# B&R Automation Studio project ControlPLC_DataDistribution (part 4)

#### Types.typ
```iecst
TYPE
	Configuration_typ : 	STRUCT
		Exists : BOOL;
		ComPortNumberZaber1Hmi : UINT;
		PyroMultiplicationFactorHmi : REAL;
	END_STRUCT;
	DI_typ : 	STRUCT
		_ : BOOL;
	END_STRUCT;
	DO_typ : 	STRUCT
		_ : BOOL;
	END_STRUCT;
	IO_typ : 	STRUCT
		do : DO_typ;
		di : DI_typ;
	END_STRUCT;
	localInterfaceCommand_typ : 	STRUCT
		exampleCommand : BOOL;
		initializeCalibration : BOOL;
		initializePixel : BOOL;
		capturePixel : BOOL;
		processPixel : BOOL;
		processCalibration : BOOL;
		uploadLUTs : BOOL;
		abort : BOOL;
		uploadTestData : BOOL;
		downloadAndParseTestResults : BOOL;
		initializeOmsTestZaber2 : BOOL;
		initializeOmsTestZaber1 : BOOL;
		setZaber1Pos : BOOL;
		setZaber2PosAndExposure : BOOL;
		checkZaber2Homed : BOOL;
		checkZaber1Homed : BOOL;
		passRequiredMetaData : BOOL;
		passCompleteHandshake : BOOL;
		passAbortedHandshake : BOOL;
		captureFrame : BOOL;
		passAbortedHandshakeWithoutAck : BOOL;
		initializePixelForFrame : BOOL;
	END_STRUCT;
	localInterfaceInternal_typ : 	STRUCT
		PLCOpen : AtnPlcOpenStatus;
		previousState : STATE;
		frameCaptured : BOOL;
		newCommand : BOOL;
		localLockout : BOOL;
		subSystemStatus : ARRAY[0..10]OF STRING[80];
		parameters : localInterfaceParameters_typ;
		missedHeartbeats : USINT;
		lastHeartbeatReceived : INT;
		calibAppNotConnected : BOOL;
		heartbeatTimer : TON;
		cmdTimeoutTimer : TON;
		cmdFrameCaptureTimer : TON;
		homeZaberWaitTimer : TON;
		moveZaberWaitTimer : TON;
		cmdZaberOnWaitTimer : TON;
		pollingAppWaitTimer : TON;
		resultsPollingTimer : TON;
		resultsTimeoutTimer : TON;
		atnPLCOpenCommandParameters : AtnPLCOpenWithParameters;
		atnPLCOpenCommand : AtnPLCOpen;
		measuredPowerList1 : ARRAY[0..100]OF REAL;
		measuredPowerList2 : ARRAY[0..100]OF REAL;
		measuredPowerList3 : ARRAY[0..100]OF REAL;
		measuredPowerList4 : ARRAY[0..100]OF REAL;
		measuredPowerList5 : ARRAY[0..100]OF REAL;
		measuredPowerList6 : ARRAY[0..100]OF REAL;
		measuredPowerList7 : ARRAY[0..100]OF REAL;
		measuredPowerList8 : ARRAY[0..100]OF REAL;
		CommandedPowerList1 : ARRAY[0..100]OF REAL;
		CommandedPowerList2 : ARRAY[0..100]OF REAL;
		CommandedPowerList3 : ARRAY[0..100]OF REAL;
		CommandedPowerList4 : ARRAY[0..100]OF REAL;
		CommandedPowerList5 : ARRAY[0..100]OF REAL;
		CommandedPowerList6 : ARRAY[0..100]OF REAL;
		CommandedPowerList7 : ARRAY[0..100]OF REAL;
		CommandedPowerList8 : ARRAY[0..100]OF REAL;
		LaserTestStatusList1 : ARRAY[0..100]OF STRING[10];
		LaserTestStatusList2 : ARRAY[0..100]OF STRING[10];
		LaserTestStatusList3 : ARRAY[0..100]OF STRING[10];
		LaserTestStatusList4 : ARRAY[0..100]OF STRING[10];
		LaserTestStatusList5 : ARRAY[0..100]OF STRING[10];
		LaserTestStatusList6 : ARRAY[0..100]OF STRING[10];
		LaserTestStatusList7 : ARRAY[0..100]OF STRING[10];
		LaserTestStatusList8 : ARRAY[0..100]OF STRING[10];
		currentPowerLevel : USINT;
		ii : USINT; (*loop variable*)
		appVersionTempString : STRING[5]; (*loop variable*)
	END_STRUCT;
	localInterfaceParameters_typ : 	STRUCT
		uploadLUTs : VFLCRUploadLUTsCmdPars_typ;
		initializePixel : VFLCRInitializePixelCmdPars_typ;
		capturePixel : VFLCRDataCollectionCmdPars_typ;
		adjustZaber1 : VFLCRAdjustZaberAndExpoPars_typ;
		adjustZaber2AndExposure : VFLCRAdjustZaberAndExpoPars_typ;
		initializePixelForFrame : VFLCRInitializePixelCmdPars_typ;
	END_STRUCT;
	localInterfaceStatus_typ : 	STRUCT
		ready : BOOL;
		state : STATE;
		sequence : SEQUENCE;
		calibAppConnected : BOOL;
		processingTestData : BOOL;
		resultsDownloaded : BOOL;
		statusMessage : STRING[vfALARMS_MAX_SNIPPET_STR_LENGTH];
		strStatus : STRING[80];
		LutIdHmi : UDINT;
		AppVersion : STRING[10];
	END_STRUCT;
	localInterface_typ : 	STRUCT
		command : localInterfaceCommand_typ;
		status : localInterfaceStatus_typ;
		internal : localInterfaceInternal_typ;
		parameters : localInterfaceParameters_typ;
	END_STRUCT;
	SEQUENCE :
		(
		SEQUENCE_IDLE,
		SEQUENCE_DONE,
		SEQUENCE_ERROR,
		SEQUENCE_LUT_DELETE,
		SEQUENCE_LUT_FTP,
		SEQUENCE_LUT_TRANSFER,
		SEQUENCE_RESULTS_DOWNLOAD,
		SEQUENCE_RESULTS_PARSE,
		SEQUENCE_MOVE_ZABER2,
		SEQUENCE_MOVE_ZABER1,
		SEQUENCE_OMS_INIT,
		SEQUENCE_OMS_ABORTED,
		SEQUENCE_WAIT_FRAME_CAPTURE
		);
	TEST_MODE :
		(
		TEST_MODE_CONTINUOUS,
		TEST_MODE_SEMI_AUTO
		);
	TEST_RESULT :
		(
		TEST_RESULT_IN_PROGRESS,
		TEST_RESULT_PASSED,
		TEST_RESULT_HIGH_POWER_FAILURE,
		TEST_RESULT_LOW_POWER_FAILURE,
		TEST_RESULT_NO_POWER_FAILURE,
		TEST_RESULT_UNTESTED,
		TEST_RESULT_ABORTED := 10
		);
	STATE :
		(
		STATE_NOT_READY,
		STATE_READY,
		STATE_DONE,
		STATE_ERROR,
		STATE_EXAMPLE_COMMAND,
		STATE_INITIALIZE_CALIBRATION,
		STATE_INITIALIZE_PIXEL,
		STATE_CAPTURE_PIXEL,
		STATE_PROCESS_PIXEL,
		STATE_PROCESS_CALIBRATION,
		STATE_UPLOAD_LUTS,
		STATE_UPLOAD_TEST_DATA,
		STATE_DOWNLOAD_PARSE_RESULTS,
		STATE_INITIALIZE_OMS_TEST_ZABER2,
		STATE_INITIALIZE_OMS_TEST_ZABER1,
		STATE_CHECK_ZABER2_HOMED,
		STATE_CHECK_ZABER1_HOMED,
		STATE_PASS_META_DATA,
		STATE_CAPTURE_FRAME,
		STATE_MOVE_ZABER2_CAM_EXPO,
		STATE_MOVE_ZABER1_CAM,
		STATE_PASS_TEST_COMPLETE,
		STATE_PASS_TEST_ABORTED,
		STATE_PASS_TEST_ABORTED_NO_ACK,
		STATE_INIT_PIXEL_FRAMECAPTURE
		);
END_TYPE
```

#### Variables.var
```iecst
VAR
	IO : IO_typ;
END_VAR
VAR RETAIN
	Configuration : Configuration_typ;
END_VAR
VAR
	task : localInterface_typ;
	logSeqChange_0 : logStateChange;
	logStateChange_0 : logStateChange;
	Name : STRING[80];
	dIn : REFERENCE TO OPCUAData_FROM_Gen3CalibApp_typ;
	dOut : REFERENCE TO OPCUAData_TO_Gen3CalibApp_typ;
	strMachineNumber : STRING[40];
	strFactoryNumber : STRING[40];
END_VAR
VAR CONSTANT
	MAX_MISSED_HEARTBEATS : USINT := 7;
END_VAR
VAR
	activePixelPlaceholder : USINT := 1;
	usingGen3LaserCalibrationApp : BOOL; (*temporary disable*)
END_VAR
```

#### Simulation.st
```iecst
ACTION SimulateIO:

END_ACTION
```

### Program Logical/ProcessControl/VFLCR/VFPTR_System (IEC)

#### Main.st - Init, cyclic, exit code
```iecst
PROGRAM _INIT

	IO.do.counterReset := TRUE;

	subscribePLCOpen(gVFLCR.command.enableModulation,  'VFPTR_System', task.command.enableModulation,  task.internal.PLCOpenEnableModulation);
	subscribePLCOpen(gVFLCR.command.disableModulation, 'VFPTR_System', task.command.disableModulation, task.internal.PLCOpenDisableModulation);

	subscribePLCOpen(gVFLCR.command.openLayer, 'VFPTR_System', task.command.pulseCounterReset, task.internal.PLCOpenCounterReset);
	subscribePLCOpen(gVFLCR.command.abortLayer, 'VFPTR_System', task.command.endTrajectory, task.internal.PLCOpenTrajectory);

	registerStateBool(gVFLCR.inhibit.autoModulation, 'VFPTR_System', task.status.counterResetEnabled);

	registerStateBool(gVFLCR.status.counterResetEnabled, 'VFPTR_System', task.status.counterResetEnabled);
	registerStateBool(gVFLCR.status.modulationEnabled, 'VFPTR_System', task.status.modulationEnabled);
	registerStateBool(gVFLCR.status.userModulationEnabled, 'VFPTR_System', task.status.userModulationEnabled);
	registerStateBool(gVFLCR.status.encoderXSelected, 'VFPTR_System', task.status.encoderXSelected);
	registerStateBool(gVFLCR.status.prepareTrajectory, 'VFPTR_System', task.status.prepareTrajectory);

	// Set timeout
	task.internal.openLayerTON.PT := T#5s;

	// Initialize the lag error statistics function block moving window length.
	FOR i := 0 TO MONITOR_AXIS_MAI BY 1 DO
		task.internal.lagErrorStatistics[i].Enable := TRUE;
		task.internal.lagErrorStatistics[i].Update := TRUE;
		task.internal.lagErrorStatistics[i].MovingWindowLength := Configuration.lagMovingAvgWindowLength;
		task.internal.lagErrorStatistics[i].In := 0.0;
		task.internal.lagErrorStatistics[i]();
	END_FOR

END_PROGRAM

PROGRAM _CYCLIC

	//PiperModuleInterface;

	// Modulation in manual mode requires:
	// - safety interlock reset
	// 		- inhibit probably set elsewhere
	// - modulationEnable flag (set by user)
	// Modulation in auto mode additionally requires:
	// - prepareTrajectory (M-flag)
	// - NOT counterReset (command, maybe also M-flag related?)
	// - build info valid
	// 		- inhibit set elsewhere
	// - CNC gantry group is in GroupStateMoving
	// 		- inhibit set elsewhere
	// - master axis homed and within build volume bounds (+/- 25mm?)
	// 		- inhibit set elsewhere

	// do.enableModulation should be TRUE only while over the build plate; other conditions apply, see above
	// do.counterReset should be FALSE while in a trajectory, TRUE otherwise. Additionally, a positive edge is required after opening a layer and before starting the first trajectory.
	// do.selectEncoderX should be TRUE while printing in the X direction and FALSE while printing in the Y direction (while not lasing, its value is benign)

	///////////////////////////////////////////////////////////////
	// API:
	//	Requires:
	//	- nothing
	//	Commands:
	//	- enableModulation 			- Allows the lasers to fire
	//	- disableModulation 		- Prevents the lasers from firing
	//  Statuses:
	//	- modulationEnabled 		- Laser modulation is currently enabled
	//	- userModulationEnabled 	- Laser modulation is currently commanded to be enabled
	//	- counterResetEnabled 		- The laser position is being forced to 0
	//	- encoderXSelected 			- The X axis is being used to determine laser position, as opposed to the Y axis
	//	- prepareTrajectory 		- A trajectory is currently being executed
	//	Inhbitits:
	//	- autoModulation 			- TODO: Set by build info, CNC gantry state, and lead axis position.
	// 									TODO: should the logic that determines which axis does the inhibiting be implemented here?
	//	- modulation 				- TODO: Set by safety interlock
	///////////////////////////////////////////////////////////////

	// Read in external components

	// Read external states
	task.status.ready := TRUE;

	task.internal.manualModeEnabled := stateAllTrue(gVFLCR.status.manualModeEnabled, TRUE);
	task.internal.laserEmissionEnabled := stateAnyTrue(gVFLCR.status.laserEmissionEnabled, FALSE);

	IF task.internal.manualModeEnabled THEN
		task.internal.modulationInhibited := TRUE;
	ELSE
		task.internal.modulationInhibited := isInhibited(gVFLCR.inhibit.modulation) OR isInhibited(gVFLCR.inhibit.autoModulation) OR NOT(task.status.prepareTrajectory) ;
	END_IF

	// Handle commands
	//IF task.command.enableModulation THEN

	//	task.status.userModulationEnabled := TRUE;
	//	gVFLCR.status.laserModulationEnabled := TRUE;
	//	task.internal.PLCOpenEnableModulation.status := ERR_OK;

//	END_IF

	IF task.command.disableModulation THEN

		task.status.userModulationEnabled := FALSE;
		task.internal.PLCOpenDisableModulation.status := ERR_OK;
		task.internal.PLCOpenEnableModulation.status := ERR_INHIBITED;

	END_IF

	IF task.command.pulseCounterReset THEN

		task.internal.newCommand := TRUE;
		task.status.state := STATE_PULSE_COUNTER_RESET;

	ELSIF task.command.beginTrajectoryX THEN

		task.internal.newCommand := TRUE;
		task.internal.setLeadX := TRUE;
		task.status.state := STATE_BEGIN_TRAJECTORY;

	ELSIF task.command.beginTrajectoryY THEN

		task.internal.newCommand := TRUE;
		task.internal.setLeadX := FALSE;
		task.status.state := STATE_BEGIN_TRAJECTORY;

	ELSIF task.command.endTrajectory THEN

		task.internal.newCommand := TRUE;
		task.status.state := STATE_READY;

	END_IF

	///////////////////////////////////////////////////////////////
	// Handle any canceled commands that are required
	///////////////////////////////////////////////////////////////
	IF task.internal.newCommand THEN

		//TODO: Log state changes
		//		task.internal.abortedStep := task.status.sequence;
		//		task.internal.abortedState := task.internal.previousState;

		task.status.sequence := SEQUENCE_IDLE;

		atnPLCOpenAbort(task.internal.PLCOpenTrajectory);
		atnPLCOpenAbort(task.internal.PLCOpenCounterReset);

	END_IF

	// Handle single-cycle commands
	IF task.command.endTrajectory THEN

		task.status.prepareTrajectory := FALSE;
		IO.do.counterReset := TRUE;
		task.internal.PLCOpenTrajectory.status := ERR_OK;

	END_IF

	///////////////////////////////////////////////////////////////
	// Handle the current state
	///////////////////////////////////////////////////////////////
	CASE task.status.state OF

		STATE_NOT_READY:

			task.status.sequence := SEQUENCE_IDLE;

			IF task.status.ready THEN

				task.status.state := STATE_READY;

			END_IF

		STATE_READY:

			task.status.sequence := SEQUENCE_IDLE;

		STATE_BEGIN_TRAJECTORY:

			CASE task.status.sequence OF
				// Non-standard sequencing to improve responsiveness
				SEQUENCE_IDLE:

					IO.do.selectEncoderX := task.internal.setLeadX;
					IO.do.counterReset := TRUE;

					IF Configuration.disableLagCheck THEN
						task.status.sequence := SEQUENCE_DONE;
					ELSE

						task.status.sequence := SEQUENCE_CHECK_LAG_IN_TOLERANCE;

					END_IF

				SEQUENCE_CHECK_LAG_IN_TOLERANCE:

					// Verify that lag error for X1 and X2 has stabilized.
					IF task.status.encoderXSelected THEN
						IF ((task.internal.lagErrorStatistics[MONITOR_AXIS_X1].Mean < Configuration.minLagToBeginTrajectory) AND
							(task.internal.lagErrorStatistics[MONITOR_AXIS_X1].StdDeviation < Configuration.minLagStdDev) AND
							(task.internal.lagErrorStatistics[MONITOR_AXIS_X2].Mean < Configuration.minLagToBeginTrajectory) AND
							(task.internal.lagErrorStatistics[MONITOR_AXIS_X2].StdDeviation < Configuration.minLagStdDev)) THEN
							task.status.sequence := SEQUENCE_DONE;
						END_IF
					// Verify that lag error for Y axis has stabilized.
					ELSE
						IF ((task.internal.lagErrorStatistics[MONITOR_AXIS_Y].Mean < Configuration.minLagToBeginTrajectory) AND
							(task.internal.lagErrorStatistics[MONITOR_AXIS_Y].StdDeviation < Configuration.minLagStdDev)) THEN
							task.status.sequence := SEQUENCE_DONE;
						END_IF
					END_IF

				SEQUENCE_DONE:

					task.status.prepareTrajectory := TRUE;
					IO.do.counterReset := FALSE;
					task.internal.PLCOpenTrajectory.status := ERR_OK;
					task.status.state := STATE_READY;

			END_CASE

		// This sequence requires the laser IO devices to check IO at least as frequently as this task runs (cycle time is currently 0.8ms)
		STATE_PULSE_COUNTER_RESET:
			// Non-standard sequencing to match STATE_BEGIN_TRAJECTORY
			CASE task.status.sequence OF

				SEQUENCE_IDLE:
					// One or more racks might fail to open layer; if so, time out instead of hanging
					task.internal.openLayerTON.IN := TRUE;

					IF stateAllTrue(gVFLCR.status.layerOpen, TRUE) THEN
						// pulse
						IO.do.counterReset := FALSE;
						task.status.sequence := SEQUENCE_DONE;

					ELSIF task.internal.openLayerTON.Q THEN
						// no need to pulse
						task.internal.PLCOpenCounterReset.status := VFLCR_ERROR;
						task.status.state := STATE_READY;

					END_IF

				SEQUENCE_DONE:

					IO.do.counterReset := TRUE;
					task.internal.PLCOpenCounterReset.status := ERR_OK;
					task.status.state := STATE_READY;

			END_CASE

	END_CASE

	///////////////////////////////////////////////////////////////
	// Reset all commands to ensure they don't get buffered
	///////////////////////////////////////////////////////////////
	brsmemset(ADR(task.command), 0, SIZEOF(task.command));
	task.internal.newCommand := FALSE;

	///////////////////////////////////////////////////////////////
	// Call all function blocks
	///////////////////////////////////////////////////////////////
	task.internal.openLayerTON();
	task.internal.openLayerTON.IN := FALSE;

	///////////////////////////////////////////////////////////////
	// Set remaining IO and statuses
	///////////////////////////////////////////////////////////////
	IO.do.enableModulation := FALSE;

	task.status.counterResetEnabled := IO.do.counterReset;
	task.status.encoderXSelected := IO.do.selectEncoderX;
	task.status.modulationEnabled := IO.do.enableModulation;

END_PROGRAM

PROGRAM _EXIT
	(* Insert code here *)

END_PROGRAM
```

### Opcua.typ
```iecst
TYPE
	OPCUAData_FROM_BuildPC_typ : 	STRUCT
		Heartbeat : UINT;
		BuildInfoReady : BOOL;
		DistributionActive : BOOL;
		DistributionPaused : BOOL;
		DistributionAborted : BOOL;
		BuildLayout : UDINT;
		PrintNumber : UINT;
		CurrentDistributionLayer : UDINT;
		StatusMessage : STRING[80];
		DataDistributorVersion : STRING[40];
	END_STRUCT;
	OPCUAData_TO_BuildPC_typ : 	STRUCT
		Heartbeat : UINT;
		RequestBuildInfo : BOOL;
		RequestStartDistribution : BOOL;
		RequestPauseDistribution : BOOL;
		RequestAbortDistribution : BOOL;
		PrintingActive : BOOL;
		CurrentPrintLayer : UDINT;
	END_STRUCT;
END_TYPE
```

### RecipeManagement.typ
```iecst
(*System Recipe*)

TYPE
	SystemRecipeManager_typ : 	STRUCT
		commands : SystemRecipeCommand_typ;
		events : SystemRecipeEvents_typ;
	END_STRUCT;
	SystemRecipeCommand_typ : 	STRUCT
		loadBuildInfo : STRING[80];
		loadCustomScanFile : STRING[80];
		loadPrintProcessConfigFile : STRING[80];
	END_STRUCT;
	SystemRecipeEvents_typ : 	STRUCT
		buildInfoLoaded : STRING[80];
		customScanLoaded : STRING[80];
	END_STRUCT;
END_TYPE

(*Single recipe handler*)
```

### Types.typ
```iecst
(*api for build distributor interface*)

TYPE
	BuildDistributor_typ : 	STRUCT
		commands : BuildDistributorCommands_typ;
		status : BuildDistributorStatus_Typ;
		alarms : BuildDistributorAlarms_typ;
	END_STRUCT;
	BuildDistributorAlarms_typ : 	STRUCT
		components : vfAlarms_Component_typ;
		BD_HEARTBEAT_LOST_AL : vfAlarms_Instance_type;
	END_STRUCT;
	BuildDistributorStatus_Typ : 	STRUCT
		subsystemsReady : STRING[80];
		isConnected : STRING[80];
	END_STRUCT;
	BuildDistributorCommands_typ : 	STRUCT
		distributeLayerFile : STRING[80];
		startDistribution : STRING[80];
		abortDistribution : STRING[80];
	END_STRUCT;
END_TYPE

(*api for print job management interface*)

TYPE
	PrintJobManagement_typ : 	STRUCT
		commands : PrintJobManagementCommands_typ;
		status : PrintJobManagementStatus_typ;
		currentState : PrintJobManagementState_typ;
		alarms : PrintJobManagementAlarms_typ;
	END_STRUCT;
	PrintJobManagementCommands_typ : 	STRUCT
		validatePrintFile : STRING[80];
		updateLayerNumber : STRING[80];
		resetPrintInfo : STRING[80];
	END_STRUCT;
	PrintJobManagementStatus_typ : 	STRUCT
		distributionLayerRecieved : BOOL;
		distributionLayerRequested : BOOL;
		buildInfoValid : STRING[80];
		buildInfoInvalid : STRING[80];
		distributionActive : BOOL;
	END_STRUCT;
	PrintJobManagementState_typ : 	STRUCT
		baseFilename : STRING[20];
		description : STRING[80];
		author : STRING[40];
		printOwner : STRING[40];
		buildInstanceID : STRING[40];
		configEditorBranch : STRING[20];
		configEditorVersion : STRING[20];
		rasterEngineBranch : STRING[20];
		rasterEngineVersion : STRING[20];
		buildLayout : UDINT;
		printNumber : UINT;
		numberOfLayers : UINT;
		currentLayerNumber : UINT;
		lastRecoatedLayerNumber : UINT;
		lastPrintedLayerNumber : UINT;
		newBuildInfoFileLoaded : BOOL;
		lastDistributedLayer : UINT;
	END_STRUCT;
	PrintJobManagementAlarms_typ : 	STRUCT
		FileLoadError_AL0023 : vfAlarms_Instance_type;
		FileSaveError_AL0024 : vfAlarms_Instance_type;
		BuildInfoValidRequired_AL0025 : vfAlarms_Instance_type;
	END_STRUCT;
END_TYPE
```

### Program Logical/ProcessControl/PrintJobManagement/BuildDistributor

#### Types.typ
```iecst
TYPE
	AI_typ : 	STRUCT
		_ : USINT;
	END_STRUCT;
	AO_typ : 	STRUCT
		_ : BOOL;
	END_STRUCT;
	DI_typ : 	STRUCT
		_ : BOOL;
	END_STRUCT;
	DO_typ : 	STRUCT
		_ : BOOL;
	END_STRUCT;
	IO_typ : 	STRUCT
		do : DO_typ;
		di : DI_typ;
	END_STRUCT;
	localInterfaceCommand_typ : 	STRUCT
		distributeLayerFile : BOOL;
		startDistribution : BOOL;
		abortDistribution : BOOL;
	END_STRUCT;
	localInterfaceInternal_typ : 	STRUCT
		PLCOpen : AtnPlcOpenStatus;
		previousState : STATE;
		newCommand : BOOL;
		localLockout : BOOL;
		subSystemStatus : ARRAY[0..10]OF STRING[80];
		lastHeartbeatReceived : INT;
		heartbeatTimer : TON;
		atnPLCOpenCommandParameters : AtnPLCOpenWithParameters;
		atnPLCOpenCommand : AtnPLCOpen;
		fbTON_DistributionDelay : TON;
		lastDistributedLayerNumber : UINT;
		waitToRetry : TON;
		retryAttempted : BOOL;
	END_STRUCT;
	localInterfaceParameters_typ : 	STRUCT
		layerNumberToDistribute : UINT;
	END_STRUCT;
	localInterfaceStatus_typ : 	STRUCT
		ready : BOOL;
		state : STATE;
		sequence : SEQUENCE;
		lastErrorState : SEQUENCE;
		buildDistributorConnected : BOOL;
		statusMessage : STRING[vfALARMS_MAX_SNIPPET_STR_LENGTH];
		missedHeartbeats : USINT;
		lastErrorMessage : STRING[40];
	END_STRUCT;
	localInterface_typ : 	STRUCT
		command : localInterfaceCommand_typ;
		status : localInterfaceStatus_typ;
		internal : localInterfaceInternal_typ;
		parameters : localInterfaceParameters_typ;
	END_STRUCT;
	SEQUENCE :
		(
		SEQUENCE_IDLE,
		SEQUENCE_DONE,
		SEQUENCE_ERROR,
		SEQUENCE_EXECUTE_START_DIST,
		SEQUENCE_CHECK_DISTRIBUTOR_READY,
		SEQUENCE_REQUEST_BUILD_INFO,
		SEQUENCE_BUILD_INFO_READY,
		SEQUENCE_LOAD_BUILD_FILE,
		SEQUENCE_CHK_BUILD_INFO_VALID,
		SEQUENCE_DELETE_LASER_FILES,
		SEQUENCE_SET_DISTRIBUTION_NUMBER,
		SEQUENCE_START_DISTRIBUTION,
		SEQUENCE_VERIFY_DISTRIBUTION,
		SEQUENCE_CALCULATE_PRINT_TIME,
		SEQUENCE_DISTRIBUTION_STARTED,
		SEQUENCE_REMAP_PIXELS,
		SEQUENCE_ENABLE_LASER_AUTO,
		SEQUENCE_LOAD_PCI_FILE,
		SEQUENCE_PUBLISH_LOAD_DATA,
		SEQUENCE_EXECUTE_GET_LAYER_FILES,
		SEQUENCE_CHK_AXES_READY,
		SEQUENCE_CHK_BUILD_INFO,
		SEQUENCE_SET_DESIRED_LAYER,
		SEQUENCE_DISTRIBUTION_DELAY,
		SEQUENCE_REQUEST_DISTRIBUTION,
		SEQUENCE_WAIT_FOR_FEEDBACK,
		SEQUENCE_RETRY_AFTER_ERROR,
		SEQUENCE_SET_CURRENT_LAYER,
		SEQUENCE_MOVE_TO_CURRENT_LAYER,
		SEQUENCE_EXECUTE_ABORT_DIST,
		SEQUENCE_CHECK_DIST_READY_ABORT,
		SEQUENCE_REQUEST_ABORT_DIST,
		SEQUENCE_WAIT_DIST_ABORTED,
		SEQUENCE_PUBLISH_ABORT_DATA
		);
	STATE :
		(
		STATE_NOT_READY,
		STATE_READY,
		STATE_DONE,
		STATE_ERROR,
		STATE_START_DISTRIBUTION,
		STATE_DISTRIBUTE_LAYER_FILE,
		STATE_ABORT_DISTRIBUTION
		);
END_TYPE
```

#### Variables.var
```iecst
VAR
	IO : IO_typ;
	task : localInterface_typ;
	logSeqChange_0 : logStateChange;
	logStateChange_0 : logStateChange;
	Name : STRING[80];
END_VAR
```

- BuildDistributorSignals.xlsx (binary file, 17163 bytes)
#### Main.st
```iecst
PROGRAM _INIT

	Name := 'Build Distributor';

	//direct commands to operate the chiller
	subscribePLCOpenWithParameters ( gBuildDistributorApi.commands.startDistribution, Name, ADR(task.parameters.layerNumberToDistribute), SIZEOF(task.parameters.layerNumberToDistribute), task.command.startDistribution, task.internal.PLCOpen);
	subscribePLCOpenWithParameters ( gBuildDistributorApi.commands.distributeLayerFile, Name, ADR(task.parameters.layerNumberToDistribute), SIZEOF(task.parameters.layerNumberToDistribute), task.command.distributeLayerFile, task.internal.PLCOpen );
	subscribePLCOpenWithParameters ( gBuildDistributorApi.commands.abortDistribution, Name, 0, 0, task.command.abortDistribution, task.internal.PLCOpen);

	//other systems can monitor this state
	registerStateBool( gBuildDistributorApi.status.subsystemsReady, Name, task.status.buildDistributorConnected);

END_PROGRAM

PROGRAM _CYCLIC

	//Call piper interface
	PiperModuleInterface;

	///////////////////////////////////////////////////////////////
	//API:
	//	Requires:
	//	-
	//	Commands:
	//	-takePrescan
	//	-takePostscan
	//  -takeManual
	//	Inhbits:
	//	-

	//  State Monitoring
	//  -
	///////////////////////////////////////////////////////////////

	//Heartbeat set and monitor
	task.internal.heartbeatTimer.PT := T#1s;
	task.internal.heartbeatTimer.IN := NOT(task.internal.heartbeatTimer.Q);
	IF (task.internal.heartbeatTimer.Q) THEN
		gOpcData_ToBuildPC.Heartbeat := gOpcData_ToBuildPC.Heartbeat + 1;
		IF (gOpcData_FromBuildPC.Heartbeat <> task.internal.lastHeartbeatReceived) THEN
			task.internal.lastHeartbeatReceived := gOpcData_FromBuildPC.Heartbeat;
			task.status.buildDistributorConnected := TRUE;
			task.status.missedHeartbeats := 0;
		ELSE
			task.status.missedHeartbeats := task.status.missedHeartbeats + 1;
			task.status.buildDistributorConnected := FALSE;
		END_IF
	END_IF
	task.internal.heartbeatTimer();

	//timeout after 3 missed heartbeats
	IF task.status.missedHeartbeats > 3 THEN
		task.status.buildDistributorConnected := FALSE;
	END_IF

	//ADD LATER TODO
	//	vfAlarmPersistent(gVisionApi.alarms.components, gVisionApi.alarms.VISION_HEARTBEAT_LOST_AL1200, NOT(task.status.visionAppConnected));

	//ready to handle commands
	task.status.ready := stateTrueStatus( gBuildDistributorApi.status.subsystemsReady, ADR(task.internal.subSystemStatus), SIZEOF(task.internal.subSystemStatus) );

	IF NOT task.status.ready THEN
		stateStatus( gBuildDistributorApi.status.subsystemsReady, ADR(task.internal.subSystemStatus), SIZEOF(task.internal.subSystemStatus) );
	ELSE
		task.internal.subSystemStatus[0] := 'Ready';
	END_IF

	///////////////////////////////////////////////////////////////
	//Handle interpreting commands that do not require STATE_READY
	///////////////////////////////////////////////////////////////
	IF task.status.ready THEN

		//NOTE: Commands that just turn ON/OFF IO CAN happen in the command translation
		IF task.command.startDistribution THEN
			task.internal.newCommand := 1;

			IF (gOpcData_FromBuildPC.BuildInfoReady) OR (gOpcData_FromBuildPC.DistributionActive) THEN
				task.status.sequence := SEQUENCE_IDLE;
				task.status.state := STATE_ABORT_DISTRIBUTION;
				task.status.statusMessage := 'Aborting Distribution';
			ELSE
				task.status.sequence := SEQUENCE_IDLE;
				task.status.state := STATE_START_DISTRIBUTION;
				task.status.statusMessage := 'Starting Distribution';
			END_IF

		ELSIF task.command.distributeLayerFile THEN
			task.internal.newCommand := 1;
			task.status.sequence := SEQUENCE_IDLE;
			task.status.state := STATE_DISTRIBUTE_LAYER_FILE;
			task.status.statusMessage := 'Distributing Layer File';

		ELSIF task.command.abortDistribution THEN
			task.internal.newCommand := 1;
			task.status.sequence := SEQUENCE_IDLE;
			task.status.state := STATE_ABORT_DISTRIBUTION;
			task.status.statusMessage := 'Aborting Distribution';

		END_IF

	ELSE
		task.internal.PLCOpen.status := BUILD_DISTRIBUTOR_ERROR;
		task.status.state := STATE_NOT_READY;
		task.internal.localLockout := FALSE;
	END_IF

	///////////////////////////////////////////////////////////////
	//Handle any canceled commands that are required
	///////////////////////////////////////////////////////////////
	IF task.internal.newCommand THEN

		//TODO: Log state changes
		//		task.internal.abortedStep := task.status.sequence;
		//		task.internal.abortedState := task.internal.previousState;

		//If a new command came into the system, abort any PLCOpen commands that were active.
		// If the command came from PLCOpen FirstPass will be true and it will not abort it
		atnPLCOpenAbort(task.internal.PLCOpen);

	END_IF

	///////////////////////////////////////////////////////////////
	//Handle any Commands that do not require state.
	///////////////////////////////////////////////////////////////

	///////////////////////////////////////////////////////////////
	//Handle the current state
	///////////////////////////////////////////////////////////////
	CASE task.status.state OF

		STATE_NOT_READY:

			task.status.sequence := SEQUENCE_IDLE;
			task.status.statusMessage := 'Build Distributor is NOT ready';
			gOpcData_ToBuildPC.RequestBuildInfo := FALSE;

			IF task.status.ready THEN
				task.status.state := STATE_READY;
				task.status.statusMessage := 'Build Distributor is ready';
			END_IF

		STATE_READY:

			task.status.sequence := SEQUENCE_IDLE;
			task.internal.localLockout := FALSE;
			gOpcData_ToBuildPC.RequestBuildInfo := FALSE;

		STATE_START_DISTRIBUTION:

			CASE task.status.sequence OF

				SEQUENCE_ERROR:
					task.status.statusMessage := 'Start Distribution ERROR';
					task.internal.PLCOpen.status := BUILD_DISTRIBUTOR_ERROR;
					task.status.state := STATE_READY;

				SEQUENCE_DONE:
					task.status.statusMessage := 'Start Distribution COMPLETE';
					task.internal.PLCOpen.status := ERR_OK;
					task.status.state := STATE_READY;

				SEQUENCE_IDLE:
					task.status.statusMessage := 'Start Distribution busy...';
					task.status.sequence := SEQUENCE_EXECUTE_START_DIST;

				ELSE

					StartDistributionSubSequence;

			END_CASE

		STATE_DISTRIBUTE_LAYER_FILE:

			CASE task.status.sequence OF

				SEQUENCE_ERROR:
					task.status.statusMessage := 'Distribute Layer ERROR';
					task.internal.PLCOpen.status := BUILD_DISTRIBUTOR_ERROR;
					task.status.state := STATE_READY;

				SEQUENCE_DONE:
					task.status.statusMessage := 'Distribute Layer COMPLETE';
					task.internal.PLCOpen.status := ERR_OK;
					task.status.state := STATE_READY;

				SEQUENCE_IDLE:
					task.status.statusMessage := 'Distribute Layer busy...';
					task.status.sequence := SEQUENCE_EXECUTE_GET_LAYER_FILES;

				ELSE

					DistributeLayerFileSubSequence;

			END_CASE

		STATE_ABORT_DISTRIBUTION:

			task.status.statusMessage := 'aborting distribution';

			IF task.status.buildDistributorConnected THEN
				//gPrint Job management files
				gOpcData_ToBuildPC.RequestAbortDistribution := TRUE;
				gOpcData_ToBuildPC.RequestPauseDistribution := FALSE;
				gOpcData_ToBuildPC.RequestStartDistribution := FALSE;
				gOpcData_ToBuildPC.PrintingActive := FALSE;
				gOpcData_ToBuildPC.RequestBuildInfo := FALSE;

			ELSE
				task.status.statusMessage := 'BD not connected';
				gOpcData_ToBuildPC.RequestAbortDistribution := FALSE;
				task.status.state := STATE_READY;
				task.internal.PLCOpen.status := ERR_OK;

			END_IF

	END_CASE

	///////////////////////////////////////////////////////////////
	//Update Statuses
	///////////////////////////////////////////////////////////////

	///////////////////////////////////////////////////////////////
	//Call all PLCOpen function blocks
	///////////////////////////////////////////////////////////////
	task.internal.fbTON_DistributionDelay();
	task.internal.fbTON_DistributionDelay.IN := FALSE;

	task.internal.atnPLCOpenCommand();
	task.internal.atnPLCOpenCommand.Execute := FALSE;

	task.internal.atnPLCOpenCommandParameters();
	task.internal.atnPLCOpenCommandParameters.Execute := FALSE;

	///////////////////////////////////////////////////////////////
	//Reset all commands to ensure they don't get buffered
	///////////////////////////////////////////////////////////////
	task.command.distributeLayerFile := 0;
	task.command.startDistribution := 0;
	task.command.abortDistribution := 0;
	task.internal.newCommand := 0;

	task.internal.waitToRetry();
	task.internal.waitToRetry.IN := FALSE;

	logStateChange_0.LoggerName := 'App';
	logStateChange_0.ModuleName := Name;
	logStateChange_0.State 		:= task.status.state;
	logStateChange_0.StateName 	:= task.status.statusMessage;
	logStateChange_0();

	logSeqChange_0.LoggerName 	:= 'App';
	logSeqChange_0.ModuleName 	:= Name;
	logSeqChange_0.State		:= task.status.sequence;
	logSeqChange_0.StateName	:= task.status.statusMessage;
	logSeqChange_0();

	//Keep track of the previous state
	task.internal.previousState := task.status.state;

	///////////////////////////////////////////////////////////////
	//Simulation
	///////////////////////////////////////////////////////////////
	IF gSimulation THEN
		SimulateIO;
	END_IF

END_PROGRAM

PROGRAM _EXIT
		(* Insert code here *)

END_PROGRAM
```

#### Simulation.st
```iecst
ACTION SimulateIO:

	IF gOpcData_ToBuildPC.RequestStartDistribution THEN

		gOpcData_FromBuildPC.DistributionActive := TRUE;
		gOpcData_FromBuildPC.CurrentDistributionLayer := gOpcData_ToBuildPC.CurrentPrintLayer;

	END_IF

	IF gOpcData_ToBuildPC.RequestAbortDistribution THEN
		gOpcData_FromBuildPC.DistributionAborted := TRUE;
		gOpcData_FromBuildPC.DistributionActive := FALSE;
	END_IF

	gOpcData_FromBuildPC.BuildInfoReady := gOpcData_ToBuildPC.RequestBuildInfo;
	gOpcData_FromBuildPC.Heartbeat := gOpcData_ToBuildPC.Heartbeat;

END_ACTION
```

#### SubSequence.st
```iecst
// Start connection to build distributor and distribute the starting files
ACTION StartDistributionSubSequence:

	CASE task.status.sequence OF

		SEQUENCE_EXECUTE_START_DIST:

			task.status.sequence := SEQUENCE_REQUEST_BUILD_INFO;

		SEQUENCE_REQUEST_BUILD_INFO:

			task.status.statusMessage := 'ask for build info file';

			//gPrint Job management files
			gOpcData_ToBuildPC.RequestAbortDistribution := FALSE;
			gOpcData_ToBuildPC.RequestPauseDistribution := FALSE;
			gOpcData_ToBuildPC.RequestStartDistribution := FALSE;
			gOpcData_ToBuildPC.PrintingActive := FALSE;
			gOpcData_ToBuildPC.RequestBuildInfo := TRUE;

			//load the last file you had saved, if its 0 get layer 1
			gOpcData_ToBuildPC.CurrentPrintLayer := gPrintJobManagement.currentState.currentLayerNumber;
			IF (gOpcData_ToBuildPC.CurrentPrintLayer = 0) THEN
				gOpcData_ToBuildPC.CurrentPrintLayer := 1;
			END_IF

			task.status.sequence := SEQUENCE_BUILD_INFO_READY;

		SEQUENCE_BUILD_INFO_READY:

			IF (gOpcData_FromBuildPC.BuildInfoReady) THEN
				gOpcData_ToBuildPC.RequestBuildInfo := FALSE;
				task.status.sequence := SEQUENCE_LOAD_PCI_FILE;
			END_IF

		SEQUENCE_LOAD_PCI_FILE:

			task.status.statusMessage := 'Loading PCI File and Verifying';

			task.internal.atnPLCOpenCommand.Command := gSystemRecipeApi.commands.loadPrintProcessConfigFile;
			task.internal.atnPLCOpenCommand.Execute := TRUE;

			IF task.internal.atnPLCOpenCommand.Done THEN
				task.status.sequence := SEQUENCE_LOAD_BUILD_FILE;
				task.internal.atnPLCOpenCommand.Execute := FALSE;

			ELSIF task.internal.atnPLCOpenCommand.Error THEN
				task.status.sequence := SEQUENCE_ERROR;
			END_IF

		SEQUENCE_LOAD_BUILD_FILE:
			task.status.statusMessage := 'load build info file';
			task.internal.atnPLCOpenCommand.Command := gSystemRecipeApi.commands.loadBuildInfo;
			task.internal.atnPLCOpenCommand.Execute := TRUE;

			IF task.internal.atnPLCOpenCommand.Done THEN
				task.status.sequence := SEQUENCE_CHK_BUILD_INFO_VALID;
				task.internal.atnPLCOpenCommand.Execute := FALSE;
			ELSIF task.internal.atnPLCOpenCommand.Error THEN
				task.status.sequence := SEQUENCE_ERROR;
			END_IF

		SEQUENCE_CHK_BUILD_INFO_VALID:
			task.status.statusMessage := 'validating build info contents';
			task.internal.atnPLCOpenCommand.Command := gPrintJobManagement.commands.validatePrintFile;
			task.internal.atnPLCOpenCommand.Execute := TRUE;

			IF task.internal.atnPLCOpenCommand.Done THEN
				task.status.sequence := SEQUENCE_DELETE_LASER_FILES;
				task.internal.atnPLCOpenCommand.Execute := FALSE;
				gPrintProcessConfigLoaded := TRUE; // Set flag after validating PCI with BuildInfo File
			ELSIF task.internal.atnPLCOpenCommand.Error THEN
				task.status.sequence := SEQUENCE_ERROR;
			END_IF

		SEQUENCE_DELETE_LASER_FILES:
			task.status.statusMessage := 'delete laser files';
			task.internal.atnPLCOpenCommand.Command := gVFLCR.command.deleteLaserControlFiles;
			task.internal.atnPLCOpenCommand.Execute := TRUE;

			IF task.internal.atnPLCOpenCommand.Done THEN
				task.status.sequence := SEQUENCE_START_DISTRIBUTION;
				task.internal.atnPLCOpenCommand.Execute := FALSE;
			ELSIF task.internal.atnPLCOpenCommand.Error THEN
				task.status.sequence := SEQUENCE_ERROR;
			END_IF

		SEQUENCE_START_DISTRIBUTION:
			task.status.statusMessage := 'distribute laser files';

			gOpcData_ToBuildPC.RequestStartDistribution := TRUE;
			task.status.sequence := SEQUENCE_VERIFY_DISTRIBUTION;

		SEQUENCE_VERIFY_DISTRIBUTION:

			task.status.statusMessage := 'verifying distribution';

			IF gOpcData_FromBuildPC.DistributionActive AND (gOpcData_FromBuildPC.CurrentDistributionLayer = gOpcData_ToBuildPC.CurrentPrintLayer) THEN
				task.internal.lastDistributedLayerNumber := UDINT_TO_UINT(gOpcData_FromBuildPC.CurrentDistributionLayer);
				gPrintJobManagement.currentState.lastDistributedLayer := task.internal.lastDistributedLayerNumber;
				task.status.sequence := SEQUENCE_SET_CURRENT_LAYER;
			END_IF

		SEQUENCE_SET_CURRENT_LAYER:

			//this is redundant, but that command also will re-set the CNC file name
			task.status.statusMessage := 'update current layer';

			//NOT NEEDED!
			task.internal.atnPLCOpenCommandParameters.Command := gPrintJobManagement.commands.updateLayerNumber;
			task.internal.atnPLCOpenCommandParameters.pParameters := ADR(task.internal.lastDistributedLayerNumber);
			task.internal.atnPLCOpenCommandParameters.sParameters := SIZEOF(task.internal.lastDistributedLayerNumber);
			task.internal.atnPLCOpenCommandParameters.Execute := TRUE;

			IF task.internal.atnPLCOpenCommandParameters.Done THEN
				task.status.sequence := SEQUENCE_DISTRIBUTION_STARTED;
				task.internal.atnPLCOpenCommandParameters.Execute := FALSE;

			ELSIF task.internal.atnPLCOpenCommandParameters.Error THEN
				task.status.sequence := SEQUENCE_ERROR;
			END_IF

		SEQUENCE_DISTRIBUTION_STARTED:
			task.status.sequence := SEQUENCE_DONE;
			gPrintJobManagement.currentState.newBuildInfoFileLoaded := TRUE;//TODO this should be set outside?

	END_CASE

END_ACTION

// Distribute Layer Files to VFLCR and adjust number
ACTION DistributeLayerFileSubSequence:

	CASE task.status.sequence OF

		SEQUENCE_EXECUTE_GET_LAYER_FILES:
			task.status.sequence := SEQUENCE_CHK_BUILD_INFO;

		SEQUENCE_CHK_BUILD_INFO:
			task.status.statusMessage := 'validating build info';
			task.internal.atnPLCOpenCommand.Command := gPrintJobManagement.commands.validatePrintFile;
			task.internal.atnPLCOpenCommand.Execute := TRUE;

			IF task.internal.atnPLCOpenCommand.Done THEN
				task.status.sequence := SEQUENCE_SET_DESIRED_LAYER;
				task.internal.atnPLCOpenCommand.Execute := FALSE;
			ELSIF task.internal.atnPLCOpenCommand.Error THEN

				task.status.lastErrorMessage := 'SEQUENCE_CHK_BUILD_INFO';
				task.status.sequence := SEQUENCE_ERROR;
			END_IF

		SEQUENCE_SET_DESIRED_LAYER:

			task.status.statusMessage := 'set layer for distribution';
			gOpcData_ToBuildPC.CurrentPrintLayer := task.parameters.layerNumberToDistribute;

			//delay for parameter to go through
			task.internal.fbTON_DistributionDelay.PT := T#0.25s;
			task.internal.fbTON_DistributionDelay.IN := TRUE;
			IF task.internal.fbTON_DistributionDelay.Q THEN
				task.status.sequence := SEQUENCE_REQUEST_DISTRIBUTION;
			END_IF

		SEQUENCE_DELETE_LASER_FILES: //is this not needed?

			task.status.statusMessage := 'delete laser control files';
			task.internal.atnPLCOpenCommand.Command := gVFLCR.command.deleteLaserControlFiles;
			task.internal.atnPLCOpenCommand.Execute := TRUE;

			IF task.internal.atnPLCOpenCommand.Done THEN
				task.status.sequence := SEQUENCE_REQUEST_DISTRIBUTION;
				task.internal.atnPLCOpenCommand.Execute := FALSE;
			ELSIF task.internal.atnPLCOpenCommand.Error THEN
				task.status.lastErrorMessage := 'SEQUENCE_DELETE_LASER_FILES';

				IF NOT(task.internal.retryAttempted) THEN
					task.status.sequence := SEQUENCE_RETRY_AFTER_ERROR;
					task.status.lastErrorState := SEQUENCE_DELETE_LASER_FILES;
				ELSE
					task.status.sequence := SEQUENCE_ERROR;
					task.internal.retryAttempted := FALSE;
				END_IF

			END_IF

		SEQUENCE_REQUEST_DISTRIBUTION:

			task.status.statusMessage := 'request distribution';
			gOpcData_ToBuildPC.PrintingActive := TRUE;
			gOpcData_ToBuildPC.RequestStartDistribution := TRUE;
			task.status.sequence := SEQUENCE_WAIT_FOR_FEEDBACK;

		SEQUENCE_WAIT_FOR_FEEDBACK:

			IF gOpcData_FromBuildPC.DistributionActive AND (gOpcData_FromBuildPC.CurrentDistributionLayer = gOpcData_ToBuildPC.CurrentPrintLayer) THEN
				task.status.sequence := SEQUENCE_SET_CURRENT_LAYER;
			END_IF

		SEQUENCE_SET_CURRENT_LAYER:

			task.status.statusMessage := 'update current layer';

			task.internal.lastDistributedLayerNumber := UDINT_TO_UINT(gOpcData_ToBuildPC.CurrentPrintLayer);
			gPrintJobManagement.currentState.lastDistributedLayer := task.internal.lastDistributedLayerNumber;

			task.internal.atnPLCOpenCommandParameters.Command := gPrintJobManagement.commands.updateLayerNumber;
			task.internal.atnPLCOpenCommandParameters.pParameters := ADR(task.internal.lastDistributedLayerNumber);
			task.internal.atnPLCOpenCommandParameters.sParameters := SIZEOF(task.internal.lastDistributedLayerNumber);
			task.internal.atnPLCOpenCommandParameters.Execute := TRUE;

			IF task.internal.atnPLCOpenCommandParameters.Done THEN
				task.status.sequence := SEQUENCE_DONE;
				task.internal.atnPLCOpenCommandParameters.Execute := FALSE;

			ELSIF task.internal.atnPLCOpenCommandParameters.Error THEN
				task.status.lastErrorMessage := 'SEQUENCE_SET_CURRENT_LAYER';

				IF NOT(task.internal.retryAttempted) THEN
					task.status.sequence := SEQUENCE_RETRY_AFTER_ERROR;
					task.status.lastErrorState := SEQUENCE_SET_CURRENT_LAYER;
				ELSE
					task.status.sequence := SEQUENCE_ERROR;
					task.internal.retryAttempted := FALSE;
				END_IF
			END_IF

		SEQUENCE_RETRY_AFTER_ERROR:

			task.internal.retryAttempted := TRUE;

			task.internal.waitToRetry.PT := T#5s;
			task.internal.waitToRetry.IN := TRUE;

			IF task.internal.waitToRetry.Q THEN
				task.status.sequence := task.status.lastErrorState;
			END_IF

	END_CASE

END_ACTION

// Abort distribution process started earlier (must be done before starting another)
ACTION AbortDistributionSubSequence:

	CASE task.status.sequence OF

		SEQUENCE_EXECUTE_ABORT_DIST:

			task.status.sequence := SEQUENCE_CHECK_DIST_READY_ABORT;

		SEQUENCE_CHECK_DIST_READY_ABORT:
			task.status.statusMessage := 'check distributor connected';
			//move this outside maybe and cyclically check for connection status and throw alarm if not connected
			IF task.status.buildDistributorConnected THEN
				task.status.sequence := SEQUENCE_REQUEST_ABORT_DIST;
			ELSE
				task.status.sequence := SEQUENCE_ERROR;
			END_IF

		SEQUENCE_REQUEST_ABORT_DIST:

			task.status.statusMessage := 'aborting distribution';

			//gPrint Job management files
			gOpcData_ToBuildPC.RequestAbortDistribution := TRUE;
			gOpcData_ToBuildPC.RequestPauseDistribution := FALSE;
			gOpcData_ToBuildPC.RequestStartDistribution := FALSE;
			gOpcData_ToBuildPC.PrintingActive := FALSE;
			gOpcData_ToBuildPC.RequestBuildInfo := FALSE;

			task.status.sequence := SEQUENCE_WAIT_DIST_ABORTED;

		SEQUENCE_WAIT_DIST_ABORTED:

			task.status.statusMessage := 'distribution aborted';

			IF (gOpcData_FromBuildPC.DistributionAborted) THEN

				gOpcData_ToBuildPC.RequestAbortDistribution := FALSE;
				task.status.sequence := SEQUENCE_DONE;
			END_IF

	END_CASE

END_ACTION
```

### Program Logical/ProcessControl/PrintJobManagement/PrintJobManagement

#### Variables.var
```iecst
VAR
	newBuildJob : BOOL := 0;
	task : localInterface_typ;
	logSeqChange_0 : logStateChange;
	logStateChange_0 : logStateChange;
	messageHandler : MessageHandler_typ;
	dCurrentState : REFERENCE TO PrintJobManagementState_typ;
	layerNumberValue_string : STRING[8] := '';
	layerNumber_string : STRING[8] := '';
	Name : STRING[80];
	auditEventString : STRING[255];
	layerFilename_GCode : STRING[255];
	currentLayerString : STRING[10];
	command : AtnPLCOpen;
END_VAR
```

#### Main.st
```iecst
PROGRAM _INIT

	Name := 'Print Job Management';

	// Restore current print job management information from permanent memory.
	gPrintJobManagement.currentState := Nonvolatile;

	gConfiguration.machineIdentity.factoryName := 'VulcanOne';
	gConfiguration.machineIdentity.machineName := 'DP13';
	gConfiguration.machineIdentity.machineNumber := 13;
	gPrintJobManagement.currentState.currentLayerNumber := 0;

	subscribePLCOpenWithParameters( gPrintJobManagement.commands.updateLayerNumber, Name, ADR(task.parameters.printJobLayer), SIZEOF(task.parameters.printJobLayer), task.command.updateCurrentLayer, task.internal.PLCOpen);

	subscribePLCOpen( gPrintJobManagement.commands.validatePrintFile, Name, task.command.validatePrintFile, task.internal.PLCOpen);

	subscribePLCOpen( gSystemRecipeApi.events.buildInfoLoaded, Name, task.command.validatePrintFile, task.internal.PLCOpen);
	subscribePLCOpen( gPrintJobManagement.commands.resetPrintInfo, Name, task.command.resetPrintInfo, task.internal.PLCOpen);
	registerStateBool( gPrintJobManagement.status.buildInfoValid, 'Build Info Loaded', task.status.buildInfoValid);

	//REASONS FOR INVALID BUILD FILE
	registerStateBool( gPrintJobManagement.status.buildInfoInvalid, 'Build Name Invalid', task.status.buildInfoInvalidReasons.invalidBuildName);
	registerStateBool( gPrintJobManagement.status.buildInfoInvalid, 'Num Layers Invalid', task.status.buildInfoInvalidReasons.invalidNumLayers);
	registerStateBool( gPrintJobManagement.status.buildInfoInvalid, 'Layer Height Invalid', task.status.buildInfoInvalidReasons.invalidLayerHeight);
	registerStateBool( gPrintJobManagement.status.buildInfoInvalid, 'Platform ID Invalid', task.status.buildInfoInvalidReasons.invalidPlatformID);
	registerStateBool( gPrintJobManagement.status.buildInfoInvalid, 'Machine Name Invalid', task.status.buildInfoInvalidReasons.invalidMachineName);
	//SIM helper for bootup to set some non vol
	IF gSimulation THEN
		//gConfiguration.machineIdentity.factoryName := 'VulcanOne';
		//gConfiguration.machineIdentity.factoryNumber := FACTORY_VULCAN_ONE;
		//gConfiguration.machineIdentity.machineGeneration := MACHINE_GENERATION_GEN3;
		//	gConfiguration.machineIdentity.machineName := 'DP13';
		//gConfiguration.machineIdentity.machineType := MACHINE_TYPE_PRINTER;
		//	gConfiguration.machineIdentity.machineNumber := 13;
		//gPrintJobManagement.currentState.currentLayerNumber := 0;

	END_IF

END_PROGRAM

PROGRAM _CYCLIC

	//Copy current state to non-volatile memory.
	Nonvolatile := gPrintJobManagement.currentState;
	dCurrentState ACCESS ADR(gPrintJobManagement.currentState);

	task.status.ready := TRUE;

	/////////////////////////////////////////////////////////////////////////////////////////////////
	//COMMANDS
	//validate build info file
	//check if ready for printing
	//increment layer number

	//Cyclically this task also manages the part height and parameters related to the build info file
	/////////////////////////////////////////////////////////////////////////////////////////////////

	IF task.status.ready THEN

		IF task.command.validatePrintFile THEN

			task.internal.newCommand := TRUE;
			task.status.statusMessage := 'Validating Build Info File';
			task.status.state := STATE_VALIDATING_BUILD_INFO;

		ELSIF task.command.updateCurrentLayer THEN

			task.internal.newCommand := TRUE;
			task.status.statusMessage := 'Updating Layer Number';
			task.status.state := STATE_UPDATE_LAYER_NUMBER;

		ELSIF task.command.resetPrintInfo THEN

			task.internal.newCommand := TRUE;
			task.status.statusMessage := 'Resetting print info';
			task.status.state := STATE_RESETTING_PRINT_INFO;

		END_IF

	ELSE

		///////////////////////////////////////////////////////////////
		// Handle any canceled commands that are required
		///////////////////////////////////////////////////////////////
		IF task.internal.newCommand THEN

			// TODO: Log state changes
			//		task.internal.abortedStep := task.status.sequence;
			//		task.internal.abortedState := task.internal.previousState;

			task.status.sequence := SEQUENCE_IDLE;

			// If a new command came into the system, abort any PLCOpen commands that were active.
			// If the command came from PLCOpen FirstPass will be true and it will not abort it
			atnPLCOpenAbort(task.internal.PLCOpen);

		END_IF

		CASE task.status.state OF

			STATE_NOT_READY:

				task.status.sequence := SEQUENCE_IDLE;

				task.status.statusMessage := 'Print job manager is not in ready state';

				IF task.status.ready THEN

					task.status.state := STATE_READY;

					task.status.statusMessage := 'Print job manager is in ready state';

				END_IF

			STATE_READY:

				task.status.sequence := SEQUENCE_IDLE;
				task.internal.localLockout := FALSE;

			STATE_RESETTING_PRINT_INFO:

				CASE task.status.sequence OF

					SEQUENCE_ERROR:
						task.status.statusMessage := 'Error resetting print data';

					//Handle Error
					task.internal.PLCOpen.status := PRINT_JOB_MANAGER_ERROR;
					task.status.state := STATE_READY;

				SEQUENCE_DONE:
					task.status.statusMessage := 'Print Data has been Reset';

					//Handle Done
					task.internal.PLCOpen.status := ERR_OK;
					task.status.state := STATE_READY;

				SEQUENCE_IDLE:

					task.status.statusMessage := 'Resetting Print Data';
					task.status.state := STATE_VALIDATING_BUILD_INFO;

				ELSE

					ResetPrintInfoSubsequence;

			END_CASE

		STATE_UPDATE_LAYER_NUMBER:
				dCurrentState.currentLayerNumber := task.parameters.printJobLayer;
				Nonvolatile.currentLayerNumber := dCurrentState.currentLayerNumber;

				// Convert the current layer number to a string with the "nnnnn" format, adding required leading 0s.
				brsitoa(dCurrentState.currentLayerNumber, ADR(layerNumberValue_string));
				IF (dCurrentState.currentLayerNumber > 9999) THEN
					layerNumber_string := '';
				ELSIF (dCurrentState.currentLayerNumber > 999) THEN
					layerNumber_string := '0';
				ELSIF (dCurrentState.currentLayerNumber > 99) THEN
					layerNumber_string := '00';
				ELSIF (dCurrentState.currentLayerNumber > 9) THEN
					layerNumber_string := '000';
				ELSE
					layerNumber_string := '0000';
				END_IF
				brsstrcat(ADR(layerNumber_string), ADR(layerNumberValue_string));

				// Format the complete layer filename for the G-code (CNC) motion control file.
				layerFilename_GCode := Nonvolatile.baseFilename;
				brsstrcat(ADR(layerFilename_GCode), ADR('_L'));
				brsstrcat(ADR(layerFilename_GCode), ADR(layerNumber_string));
				brsstrcat(ADR(layerFilename_GCode), ADR('_GCode.cnc'));
				task.status.currentLayerGCodeFilename := layerFilename_GCode;

				task.internal.PLCOpen.status := ERR_OK;
				task.status.state := STATE_READY;

		STATE_VALIDATING_BUILD_INFO:

			CASE task.status.sequence OF

				SEQUENCE_ERROR:
					task.status.statusMessage := 'Error Validating Print Files';

					//Handle Error
					task.internal.PLCOpen.status := PRINT_JOB_MANAGER_ERROR;
					task.status.state := STATE_READY;

				SEQUENCE_DONE:
					task.status.statusMessage := 'Pre-Scan imaging sequence finished';

					//Handle Done
					task.internal.PLCOpen.status := ERR_OK;
					task.status.state := STATE_READY;

				SEQUENCE_IDLE:

					task.status.statusMessage := 'Pre-Scan sequence started';
					task.internal.PLCOpen.status := ERR_OK;
					task.status.state := STATE_READY;

				ELSE

					ValidateBuildFileSubsequence;

			END_CASE

		END_CASE
	END_IF

		//Set Nonvolatile cyclically
		Nonvolatile.lastRecoatedLayerNumber := dCurrentState.lastRecoatedLayerNumber;
		Nonvolatile.lastPrintedLayerNumber := dCurrentState.lastPrintedLayerNumber;

		//RESET COMMANDS
		brsmemset(ADR(task.command), 0, SIZEOF(task.command));
		task.internal.newCommand := FALSE;

		task.internal.newCommand := 0;

		command();
		IF command.Done OR command.Error OR command.Aborted THEN
			command.Execute := FALSE;
		END_IF

		logStateChange_0.LoggerName := 'App';
		logStateChange_0.ModuleName := Name;
		logStateChange_0.State 		:= task.status.state;
		logStateChange_0.StateName 	:= task.status.statusMessage;
		logStateChange_0();

		logSeqChange_0.LoggerName 	:= 'App';
		logSeqChange_0.ModuleName 	:= Name;
		//	logSeqChange_0.State		:= task.status.sequence;
		//	logSeqChange_0.StateName	:= task.status.statusMessage;
		//	logSeqChange_0();

		// ---------------------------------------------------------------------------
		// Call ATN FUB
		// ---------------------------------------------------------------------------

		task.status.buildInfoValid := stateAllFalse( gPrintJobManagement.status.buildInfoInvalid, TRUE);

		END_PROGRAM

		PROGRAM _EXIT

		END_PROGRAM
```

#### SubSequence.st
```iecst
ACTION ValidateBuildFileSubsequence:

	CASE task.status.sequence OF

		SEQUENCE_READ_BUILD_INFO:

			task.status.statusMessage := 'Checking build info contents';

			// NOTES:====================================================
			// base_filename must be 13 charaters long (e.g. VF-00001-0001)
			// build_layout and print_number must be > 0
			// num_layers must be > 0
			// layer_height must be within established range
			// PLATFORM_MEDIUM_400x600 is not currently supported
			// PrinterInfo.name must match the machineIdentity.machineName setting

			task.status.buildInfoInvalidReasons.invalidBuildName := (gBuildInformation.build_layout = 0) OR (gBuildInformation.print_number = 0) OR (brsstrlen(ADR(gBuildInformation.base_filename)) <> 13);
			task.status.buildInfoInvalidReasons.invalidNumLayers := (gBuildInformation.num_layers = 0);
			task.status.buildInfoInvalidReasons.invalidLayerHeight := (gBuildInformation.layer_height < MIN_LAYER_HEIGHT) OR (gBuildInformation.layer_height > MAX_LAYER_HEIGHT);

			IF stateAnyTrue(gPrintJobManagement.status.buildInfoInvalid, FALSE) THEN
				task.status.buildInfoValid := FALSE;
				task.status.currentLayerGCodeFilename := '';
				//get reason
				task.status.buildInfoError := stateTrueStatus( gPrintJobManagement.status.buildInfoInvalid, ADR( task.status.buildInfoErrorStatus ), SIZEOF(task.status.buildInfoErrorStatus));

				//alarm with reason
				//vfAlarmEdgeSnippet( gPrintJobManagement.alarms.components, gPrintJobManagement.alarms.BuildInfoFileError_AL0020, task.status.buildInfoErrorStatus[0]);

				task.status.sequence := SEQUENCE_ERROR;
			ELSE
				task.status.buildInfoValid := TRUE;
				// If the BuildInfo file is different from the one that was previously running, reset to layer zero to start a new print.
				(*	IF (gBuildInformation.build_layout <> dCurrentState.buildLayout)
				OR (gBuildInformation.print_number <> dCurrentState.printNumber)
				OR (gBuildInformation.layer_height <> dCurrentState.layerHeight) THEN

				task.command.resetLayerNumberToZero := TRUE;//todo
				ELSE *)

				//populate print info
				dCurrentState.baseFilename := gBuildInformation.base_filename;
				//dCurrentState.buildIteration := gBuildInformation.build_iter;
				dCurrentState.buildLayout := gBuildInformation.build_layout;
				dCurrentState.printNumber := gBuildInformation.print_number;
				dCurrentState.numberOfLayers := gBuildInformation.num_layers;
				//dCurrentState.layerHeight := gBuildInformation.layer_height;
				//dCurrentState.buildPlatform := PLATFORM_LARGE_600x600;//fixed value ignore BD
				dCurrentState.description := gBuildInformation.description;
				dCurrentState.author := gBuildInformation.author;
				dCurrentState.printOwner := gBuildInformation.print_owner;
				//dCurrentState.buildPlatformName := gBuildInformation.platform_name;
				//dCurrentState.buildVolumeExtents := gBuildInformation.build_volume_limits;
				//dCurrentState.pixelMapFileVersion := gBuildInformation.BuildInstanceInfo.PrinterInfo.vfpmap_version;
				dCurrentState.buildInstanceID := gBuildInformation.BuildInstanceInfo.base_unique_id;
				//dCurrentState.encoderTickWidth := gBuildInformation.BuildInstanceInfo.PrinterInfo.encoder_tick_width;
				//dCurrentState.maxLaserCount := gBuildInformation.BuildInstanceInfo.PrinterInfo.max_laser_count;
			//dCurrentState.laserLineAngle := gBuildInformation.BuildInstanceInfo.PrinterInfo.laser_line_angle;
				//dCurrentState.headCenterOffset := gBuildInformation.BuildInstanceInfo.PrinterInfo.head_center_offset;
				//dCurrentState.laserSpacing := gBuildInformation.BuildInstanceInfo.PrinterInfo.laser_spacing;
				//dCurrentState.minLaserWatts := gBuildInformation.BuildInstanceInfo.PrinterInfo.min_laser_watts;
				//dCurrentState.maxLaserWatts := gBuildInformation.BuildInstanceInfo.PrinterInfo.max_laser_watts;

				// If no description is provided, use the build instance ID as the description (for display on top status bar).
				IF (dCurrentState.description = '') THEN
					dCurrentState.description := dCurrentState.buildInstanceID;
				END_IF

				dCurrentState.configEditorBranch := gBuildInformation.SoftwareInfo.Configuration_Editor.branch;
				dCurrentState.configEditorVersion := gBuildInformation.SoftwareInfo.Configuration_Editor.version;
				dCurrentState.rasterEngineBranch := gBuildInformation.SoftwareInfo.Raster_Engine.branch;
				dCurrentState.rasterEngineVersion := gBuildInformation.SoftwareInfo.Raster_Engine.version;

				// Save current job info in permanent memory.
				Nonvolatile.baseFilename := dCurrentState.baseFilename;
				//Nonvolatile.buildIteration := dCurrentState.buildIteration;
				Nonvolatile.buildLayout := dCurrentState.buildLayout;
				Nonvolatile.printNumber	:= dCurrentState.printNumber;
				Nonvolatile.numberOfLayers := dCurrentState.numberOfLayers;
				//Nonvolatile.layerHeight := dCurrentState.layerHeight;
				//Nonvolatile.buildPlatform := dCurrentState.buildPlatform;
				Nonvolatile.description := dCurrentState.description;
				Nonvolatile.author := dCurrentState.author;
				Nonvolatile.printOwner := dCurrentState.printOwner;
				//Nonvolatile.buildPlatformName := dCurrentState.buildPlatformName;
				//Nonvolatile.buildVolumeExtents := dCurrentState.buildVolumeExtents;
				//Nonvolatile.pixelMapFileVersion := dCurrentState.pixelMapFileVersion;
				//Nonvolatile.buildInstanceID := dCurrentState.buildInstanceID;
				//Nonvolatile.configEditorBranch := dCurrentState.configEditorBranch;
			//	Nonvolatile.configEditorVersion := dCurrentState.configEditorVersion;
				//Nonvolatile.rasterEngineBranch := dCurrentState.rasterEngineBranch;
			//	Nonvolatile.rasterEngineVersion := dCurrentState.rasterEngineVersion;
			//	Nonvolatile.encoderTickWidth := dCurrentState.encoderTickWidth;
			//	Nonvolatile.maxLaserCount := dCurrentState.maxLaserCount;
			//	Nonvolatile.laserLineAngle := dCurrentState.laserLineAngle;
			//	Nonvolatile.headCenterOffset := dCurrentState.headCenterOffset;
			//	Nonvolatile.laserSpacing := dCurrentState.laserSpacing;
			//	Nonvolatile.minLaserWatts := dCurrentState.minLaserWatts;
			//	Nonvolatile.maxLaserWatts := dCurrentState.maxLaserWatts;

				task.status.sequence := SEQUENCE_DONE;

			END_IF

	END_CASE

END_ACTION

ACTION ResetPrintInfoSubsequence:

	CASE task.status.sequence OF

		SEQUENCE_ABORT_DISTRIBUTION:

			executeCommand(gBuildDistributorApi.commands.abortDistribution);
			task.status.sequence := SEQUENCE_CLEAR_DATA;

		SEQUENCE_CLEAR_DATA:

			dCurrentState.lastRecoatedLayerNumber := 0;
			dCurrentState.lastPrintedLayerNumber := 0;
			dCurrentState.author := '';
			dCurrentState.baseFilename := '';
			dCurrentState.buildInstanceID := '';
			dCurrentState.numberOfLayers := 0;
			task.status.sequence := SEQUENCE_DONE;
		END_CASE

	END_ACTION
```

### Program Logical/ProcessControl/PrintJobManagement/RM_BuildInfo

#### Types.typ
```iecst
TYPE
	RecipeFile_typ : 	STRUCT
		commands : RecipeCommands_typ;
		parameters : RecipeParameters_typ;
		status : RecipeStatus_typ;
		internal : RecipeInternal_typ;
	END_STRUCT;
	RecipeCommands_typ : 	STRUCT
		load : BOOL;
		save : BOOL;
	END_STRUCT;
	RecipeParameters_typ : 	STRUCT
		_ : STRING[260];
	END_STRUCT;
	RecipeStatus_typ : 	STRUCT
		state : STATE;
		busy : BOOL;
		done : BOOL;
		error : BOOL;
		errorId : DINT;
	END_STRUCT;
	RecipeInternal_typ : 	STRUCT
		save : AtnPlcOpenStatus;
		load : AtnPlcOpenStatus;
		notLoaded : BOOL;
		loaded : STRING[80];
	END_STRUCT;
	STATE :
		(
		STATE_NOT_READY,
		STATE_READY,
		STATE_DONE,
		STATE_ERROR,
		STATE_LOAD,
		STATE_SAVE
		);
END_TYPE
```

#### Variables.var
```iecst
VAR
	saveTime : DATE_AND_TIME := DT#1970-01-01-00:00:00;
	fbDTGetTime : DTGetTime := (0);
	header_MachineSettings : MpRecipeXmlHeaderType := (0);
	fbRecipeRegPar_MachineSettings : MpRecipeRegPar := (0);
	fbRecipeXml_MachineSettings : MpRecipeXml := (0);
	fbRecipeRegPar_BuildInfo : MpRecipeRegPar := (0);
	fbRecipeXml_BuildInfo : MpRecipeXml := (0);
	task : RecipeFile_typ;
END_VAR
```

#### Main.st
```iecst
PROGRAM _INIT

	//gOpcData_ToBuildPC.Heartbeat := 0;
	//gOpcData_FromBuildPC.Heartbeat := 0;

	//gOpcData_ToVisionPC.HeartbeatOut := 0;
	//gOpcData_FromVisionPC.HeartbeatIn := 0;

	gBuildInformation.base_filename := 'VF-99999-9999';
	gBuildInformation.build_iter := 0;
	gBuildInformation.description := 'n/a';
	gBuildInformation.build_layout := 99999;
	gBuildInformation.print_number := 9999;
	gBuildInformation.num_layers := 1;
	gBuildInformation.layer_height := 0.05;
	gBuildInformation.platform_id := 3;
	gBuildInformation.description := '';
	gBuildInformation.author := '';
	gBuildInformation.print_owner := '';
	gBuildInformation.platform_name := '600x600';

	subscribePLCOpen( gSystemRecipeApi.commands.loadBuildInfo, 'Build Info', task.commands.load, task.internal.load );

	task.internal.loaded := gSystemRecipeApi.events.buildInfoLoaded;

	registerStateBool( gPrintJobManagement.status.buildInfoInvalid, 'File Not Loaded', task.internal.notLoaded);

	task.internal.notLoaded := TRUE;

END_PROGRAM

PROGRAM _CYCLIC

	// Get the current date/time for save operations.
	fbDTGetTime.enable := TRUE;
	fbDTGetTime();
	saveTime := fbDTGetTime.DT1;

	// ---------------------------------------------------------------------------
	// BuildInfo recipe file management.
	// ---------------------------------------------------------------------------
	IF task.status.state = STATE_READY THEN

		// Prevent simultaneous load and save commands.
		//If both are true, cancel them both..
		IF (task.commands.load AND task.commands.save) THEN

			//task.internal.save.status := ERR_INHIBITED;
			//task.internal.load.status := ERR_INHIBITED;

			//vfAlarmEdgeSnippet( gPrintJobManagement.alarms.components, gPrintJobManagement.alarms.Inhibited_AL0022, 'Load and Save commanded at the same time');

		ELSIF task.commands.load THEN

			task.commands.load := FALSE;
			task.status.state:= STATE_LOAD;

		ELSIF task.commands.save THEN

			task.commands.save := FALSE;
			task.status.state:= STATE_SAVE;

		END_IF
	ELSE

		//TODO: Should we allow this?
		//Respond error to commands that come in while we are busy
		//Currently, this will allow commands to be saved
		//and processed when they are complete
		IF task.commands.load THEN
//			task.internal.load.status := ERR_INHIBITED;
		END_IF

		IF task.commands.load THEN
//			task.internal.save.status := ERR_INHIBITED;
		END_IF

	END_IF

	CASE task.status.state OF
		STATE_LOAD:

			fbRecipeXml_BuildInfo.Load := TRUE;

			IF fbRecipeXml_BuildInfo.CommandDone THEN

				task.internal.notLoaded := FALSE;
				task.status.state := STATE_READY;
				task.internal.load.status := ERR_OK;

				executeCommand( task.internal.loaded );

			ELSIF fbRecipeXml_BuildInfo.Error THEN

				task.internal.notLoaded := TRUE;

				fbRecipeXml_BuildInfo.ErrorReset	:= TRUE;
				task.internal.load.status := PRINT_JOB_MANAGER_ERROR;
				task.status.state := STATE_READY;

				//brsitoa(fbRecipeXml_BuildInfo.StatusID, ADR(gPrintJobManagement.alarms.FileLoadError_AL0023.snippet));
				//vfAlarmEdge( gPrintJobManagement.alarms.components, gPrintJobManagement.alarms.FileLoadError_AL0023);

			END_IF

		STATE_SAVE:

			fbRecipeXml_BuildInfo.Save := TRUE;

			IF fbRecipeXml_BuildInfo.CommandDone THEN

				task.status.state := STATE_READY;
				task.internal.save.status := ERR_OK;

			ELSIF fbRecipeXml_BuildInfo.Error THEN

				fbRecipeXml_BuildInfo.ErrorReset	:= TRUE;
				task.internal.save.status := PRINT_JOB_MANAGER_ERROR;
				task.status.state := STATE_READY;

				//brsitoa( fbRecipeXml_BuildInfo.StatusID, ADR(gPrintJobManagement.alarms.FileSaveError_AL0024.snippet));
				//vfAlarmEdge( gPrintJobManagement.alarms.components, gPrintJobManagement.alarms.FileSaveError_AL0024);

			END_IF

	END_CASE

	fbRecipeXml_BuildInfo.MpLink := ADR(gBuildInfoRecipe);
	fbRecipeXml_BuildInfo.Enable := TRUE;
	fbRecipeXml_BuildInfo.DeviceName := ADR('CurrentBuild');
	fbRecipeXml_BuildInfo.Category := ADR('BuildInfo');
	fbRecipeXml_BuildInfo.FileName := ADR('BuildInfo.xml');
	//fbRecipeXml_BuildInfo.Header := ADR(header_BuildInfo);  // BuildInfo.xml file has no header
	fbRecipeXml_BuildInfo.LoadType := mpRECIPE_XML_LOAD_ALL;
	fbRecipeXml_BuildInfo();
	fbRecipeXml_BuildInfo.Save := FALSE;
	fbRecipeXml_BuildInfo.Load := FALSE;
	fbRecipeXml_BuildInfo.ErrorReset := FALSE;

	fbRecipeRegPar_BuildInfo.MpLink := ADR(gBuildInfoRecipe);
	fbRecipeRegPar_BuildInfo.Enable := TRUE;
	fbRecipeRegPar_BuildInfo.PVName := ADR('gBuildInformation');
	fbRecipeRegPar_BuildInfo.Category := ADR('BuildInfo');
	fbRecipeRegPar_BuildInfo();
	fbRecipeRegPar_BuildInfo.ErrorReset := FALSE;

	//If we are not ready, and the build info IS ready, go to ready
	IF task.status.state =  STATE_NOT_READY AND fbRecipeRegPar_BuildInfo.StatusID = ERR_OK THEN

		task.status.state:= STATE_READY;

	END_IF

	// Update the command status; if an error occurs, update select the first applicable status ID.
	task.status.busy := fbRecipeXml_BuildInfo.CommandBusy;
	task.status.done := fbRecipeXml_BuildInfo.CommandDone;
	task.status.error := fbRecipeRegPar_BuildInfo.Error OR fbRecipeXml_BuildInfo.Error;
	IF (fbRecipeRegPar_BuildInfo.Error) THEN
		task.status.errorId := fbRecipeRegPar_BuildInfo.StatusID;
	ELSIF (fbRecipeXml_BuildInfo.Error) THEN
		task.status.errorId := fbRecipeXml_BuildInfo.StatusID;
	ELSE
		task.status.errorId := ERR_OK;
	END_IF

END_PROGRAM

PROGRAM _EXIT

	// Prevent error mpRECIPE_ERR_MPLINK_IN_USE by releasing the link to the configuration objects.
	fbRecipeRegPar_BuildInfo.Enable := FALSE;
	fbRecipeRegPar_BuildInfo();
	fbRecipeXml_BuildInfo.Enable := FALSE;
	fbRecipeXml_BuildInfo();

END_PROGRAM
```

### Program Logical/ProcessControl/PrintJobManagement/RM_PrintProcessConfig

#### Cyclic.st
```iecst
PROGRAM _CYCLIC

	// ---------------------------------------------------------------------------
	// PrintProcessConfig recipe file management.
	// ---------------------------------------------------------------------------

	IF task.status.state = STATE_READY THEN

		IF  task.commands.load THEN

			task.status.state:= STATE_LOAD;

		END_IF

	ELSE

		//TODO: Should we allow this?
		//Respond error to commands that come in while we are busy
		//Currently, this will allow commands to be saved
		//and processed when they are complete
		IF task.commands.load THEN
			//			task.internal.load.status := ERR_INHIBITED;
		END_IF

		IF task.commands.load THEN
			//			task.internal.save.status := ERR_INHIBITED;
		END_IF

	END_IF

	CASE task.status.state OF

		STATE_LOAD:

			fbRecipeXml_PrintProcessConfig.Load := TRUE;

			IF fbRecipeXml_PrintProcessConfig.CommandDone THEN

				task.internal.load.status := ERR_OK;

				task.status.state := STATE_READY;

			ELSIF fbRecipeXml_PrintProcessConfig.Error THEN

				fbRecipeXml_PrintProcessConfig.ErrorReset	:= TRUE;
				task.internal.load.status := PRINT_JOB_MANAGER_ERROR;

				task.status.state := STATE_READY;

				//brsitoa(fbRecipeXml_PrintProcessConfig.StatusID, ADR(gPrintJobManagement.alarms.FileLoadError_AL0023.snippet));
				//vfAlarmEdge( gPrintJobManagement.alarms.components, gPrintJobManagement.alarms.FileLoadError_AL0023);

			END_IF

		STATE_SAVE:

			fbRecipeXml_PrintProcessConfig.Save := TRUE;

			IF fbRecipeXml_PrintProcessConfig.CommandDone THEN

				task.status.state := STATE_READY;
				task.internal.save.status := ERR_OK;

			ELSIF fbRecipeXml_PrintProcessConfig.Error THEN

				fbRecipeXml_PrintProcessConfig.ErrorReset	:= TRUE;
				task.internal.save.status := PRINT_JOB_MANAGER_ERROR;
				task.status.state := STATE_READY;

				//brsitoa( fbRecipeXml_PrintProcessConfig.StatusID, ADR(gPrintJobManagement.alarms.FileSaveError_AL0024.snippet));
				//vfAlarmEdge( gPrintJobManagement.alarms.components, gPrintJobManagement.alarms.FileSaveError_AL0024);

			END_IF

	END_CASE

	task.commands.load := FALSE;
	task.commands.save := FALSE;

	//If we are not ready, and the build info IS ready, go to ready
	IF task.status.state =  STATE_NOT_READY AND fbRecipeRegPar_PrintConfig.StatusID = ERR_OK THEN

		task.status.state:= STATE_READY;

	END_IF

	// Update the command status; if an error occurs, update select the first applicable status ID.
	task.status.busy := fbRecipeXml_PrintProcessConfig.CommandBusy;
	task.status.done := fbRecipeXml_PrintProcessConfig.CommandDone;
	task.status.error := fbRecipeRegPar_PrintConfig.Error OR fbRecipeXml_PrintProcessConfig.Error;
	IF (fbRecipeRegPar_PrintConfig.Error) THEN
		task.status.errorId := fbRecipeRegPar_PrintConfig.StatusID;
	ELSIF (fbRecipeXml_PrintProcessConfig.Error) THEN
		task.status.errorId := fbRecipeXml_PrintProcessConfig.StatusID;
	ELSE
		task.status.errorId := ERR_OK;

	END_IF

	DeriveProcessData;

END_PROGRAM
```

#### DeriveProcessData.st
```iecst
ACTION DeriveProcessData:

	// ==================================================================================================================================================

	IF gPrintProcessConfigLoaded THEN
		task.status.pciLoadStatus := 'LOADED';
	ELSE
		task.status.pciLoadStatus := 'NOT LOADED';
	END_IF

END_ACTION
```

#### Init.st
```iecst
PROGRAM _INIT

	subscribePLCOpen( gSystemRecipeApi.commands.loadPrintProcessConfigFile, 'Print Process Config File Load', task.commands.load, task.internal.load );

END_PROGRAM
```

### BuildInformation.typ
```iecst
TYPE
	BuildCoordinate_typ : 	STRUCT
		X : REAL;
		Y : REAL;
		Z : REAL;
	END_STRUCT;
	BuildVolumeExtents_typ : 	STRUCT
		min : BuildCoordinate_typ;
		max : BuildCoordinate_typ;
	END_STRUCT;
	BuildInformation_typ : 	STRUCT  (*CAUTION: Structure member names must match those in BuildInfo.xml file*)
		base_filename : STRING[20]; (*example:  VF-XXXXX-YYYY*)
		build_iter : UINT; (*example:  2*)
		build_layout : UDINT; (*example:  XXXXX*)
		print_number : UINT; (*example:  YYYY*)
		num_layers : UINT; (*example:  1000*)
		layer_height : REAL; (*example:  0.050*)
		num_trajectories_x : UDINT;
		num_trajectories_y : UDINT;
		num_intralayer_gashead_cleans : UINT;
		avg_trajectory_length_y : REAL;
		total_cooling_delay : UDINT;
		avg_trajectory_length_x : REAL;
		trajectory_velocity : REAL;
		trajectory_acceleration : REAL;
		index_velocity : REAL;
		index_acceleration : REAL;
		platform_id : USINT; (*example:  1=200x600, 2=400x600, 3=600x600, 4=...*)
		description : STRING[80]; (*example:  ZStepFocusTest*)
		author : STRING[40]; (*example:  Joe Schmoe*)
		print_owner : STRING[40]; (*example:  Joe Schmoe*)
		platform_name : STRING[20]; (*example:  200x600*)
		cmmFilename : STRING[100];
		CameraCalibration : UINT;
		SubPlateInUse : BOOL;
		build_volume_limits : BuildVolumeExtents_typ;
		SoftwareInfo : BuildSoftwareInfo_typ;
		BuildInstanceInfo : BuildInstanceInfo_typ;
		BuildPrinterInfo : BuildPrinterInfo_typ;
	END_STRUCT;
	BuildInstanceInfo_typ : 	STRUCT
		base_unique_id : STRING[40]; (*example:  2021-08-27-08-59-55-VF-00244-0007*)
		PrinterInfo : BuildPrinterInfo_typ;
		active_pixels : ARRAY[0..147]OF BOOL; (*example:  pixel number is TRUE if used by the build, FALSE if not used*)
	END_STRUCT;
	BuildPrinterInfo_typ : 	STRUCT
		name : STRING[20]; (*example:  BETA, GEN2, DP1, DP2, ... DP21*)
		vfpmap_version : UINT; (*example:  3*)
		encoder_tick_width : REAL; (*example:  0.001000*)
		max_gantry_speed : REAL; (*example:  1000*)
		max_gantry_acceleration : REAL; (*example:  9800*)
		max_laser_count : UINT; (*example:  147*)
		laser_line_angle : REAL; (*example:  45.00*)
		head_center_offset : REAL; (*example:  36.750*)
		laser_spacing : REAL; (*example:  0.500*)
		min_laser_watts : REAL; (*example:  0*)
		max_laser_watts : REAL; (*example:  525*)
		phy_laser_encoding : STRING[20]; (*example:  VFLCR*)
		gantry_max_pos_x : REAL;
		gantry_max_pos_y : REAL;
		gantry_min_pos_x : REAL;
		gantry_min_pos_y : REAL;
	END_STRUCT;
	BuildSoftwareInfoDetails_typ : 	STRUCT
		version : STRING[20]; (*example:  1_2_8*)
		branch : STRING[20]; (*example:  master*)
		commit : STRING[60]; (*example:  814c89354298fdffd768bf74d4408e2ac6ac2c64*)
	END_STRUCT;
	BuildSoftwareInfo_typ : 	STRUCT
		Configuration_Editor : BuildSoftwareInfoDetails_typ;
		Raster_Engine : BuildSoftwareInfoDetails_typ;
	END_STRUCT;
END_TYPE

(*PRINT PROCESS CONFIG*)

TYPE
	PrintProcessConfig_typ : 	STRUCT
		MachineName : STRING[5];
		Description : STRING[255];
		FileFormatVersion : INT;
		DateTimeGenerated : STRING[30];
		ParamterSetpoints : ARRAY[1..DIGITAL_PCI_MAX_PARS]OF ParamterSetpoints_typ;
	END_STRUCT;
	ParamterSetpoints_typ : 	STRUCT
		Name : STRING[50];
		Used : BOOL;
		EngineeringUnits : STRING[25];
		ParDataType : STRING[10];
		HmiRangeMin : REAL;
		HmiRangeMax : REAL;
		FixedValue : REAL;
		EnableLayerRangeChanges : BOOL;
		NumberOfLayerValuesUsed : USINT;
		LayerSpecificValues : ARRAY[1..DIGITAL_PCI_MAX_LAYER_CHANGE]OF LayerSpecificValues_typ;
	END_STRUCT;
	LayerSpecificValues_typ : 	STRUCT
		LayerValue : REAL;
		LayerStart : INT;
		LayerEnd : INT;
	END_STRUCT;
	DerivedProcessParameters_typ : 	STRUCT
		Name : STRING[50];
		Used : BOOL;
		EngineeringUnits : STRING[25];
		ParDataType : STRING[10];
		HmiRangeMin : REAL;
		HmiRangeMax : REAL;
		DerivedValue : REAL;
	END_STRUCT;
	ProcessParameters :
		(
		CONTINUOUS_MODE_ENABLE := 1,
		GAS_FLOW_LPM,
		REC_SPREAD_MOVE_VEL,
		REC_APPROACH_MOVE_VEL,
		ELECTRODE_ENABLE,
		ELECTRODE_GAIN_PERCENT,
		MH_INITIAL_DISP_ROTATIONS,
		MH_CONT_DISP_ROTATIONS,
		AI_MAX_RECOAT_LIMIT
		);
END_TYPE
```

### RecipeManagement.typ
```iecst
(*System Recipe*)

TYPE
	SystemRecipeManager_typ : 	STRUCT
		commands : SystemRecipeCommand_typ;
		status : SystemRecipeStatus_typ;
		events : SystemRecipeEvents_typ;
	END_STRUCT;
	SystemRecipeCommand_typ : 	STRUCT
		loadBuildInfo : STRING[80];
		loadCustomScanFile : STRING[80];
		loadPrintProcessConfigFile : STRING[80];
	END_STRUCT;
	SystemRecipeStatus_typ : 	STRUCT
		buildInfoLoaded : BOOL;
	END_STRUCT;
	SystemRecipeEvents_typ : 	STRUCT
		buildInfoLoaded : STRING[80];
		customScanLoaded : STRING[80];
	END_STRUCT;
END_TYPE

(*Single recipe handler*)
```

### Types.typ
```iecst
(*api for build distributor interface*)

TYPE
	BuildDistributor_typ : 	STRUCT
		commands : BuildDistributorCommands_typ;
		status : BuildDistributorStatus_Typ;
		alarms : BuildDistributorAlarms_typ;
	END_STRUCT;
	BuildDistributorAlarms_typ : 	STRUCT
		components : vfAlarms_Component_typ;
		BD_HEARTBEAT_LOST_AL : vfAlarms_Instance_type;
	END_STRUCT;
	BuildDistributorStatus_Typ : 	STRUCT
		subsystemsReady : STRING[80];
		isConnected : STRING[80];
	END_STRUCT;
	BuildDistributorCommands_typ : 	STRUCT
		distributeLayerFile : STRING[80];
		startDistribution : STRING[80];
		abortDistribution : STRING[80];
	END_STRUCT;
	BuildPlatform_enum :
		(
		PLATFORM_UNKNOWN := 0,
		PLATFORM_SMALL_200x600 := 1,
		PLATFORM_MEDIUM_400x600 := 2,
		PLATFORM_LARGE_600x600 := 3
		);
END_TYPE

(*api for print job management interface*)

TYPE
	PrintJobManagement_typ : 	STRUCT
		commands : PrintJobManagementCommands_typ;
		status : PrintJobManagementStatus_typ;
		currentState : PrintJobManagementState_typ;
	END_STRUCT;
	PrintJobManagementCommands_typ : 	STRUCT
		validatePrintFile : STRING[80];
		updateLayerNumber : STRING[80];
		resetPrintInfo : STRING[80];
		enableLOP : STRING[80];
		disableLOP : STRING[80];
	END_STRUCT;
	PrintJobManagementStatus_typ : 	STRUCT
		distributionLayerRecieved : BOOL;
		distributionLayerRequested : BOOL;
		loadPCIFileComplete : BOOL;
		distributionLayerComplete : BOOL;
		buildInfoValidCheck : BOOL;
		buildInfoValid : STRING[80];
		currentLayerGCodeFilename : STRING[255];
		buildInfoInvalid : STRING[80];
		distributionActive : BOOL;
	END_STRUCT;
	PrintJobManagementState_typ : 	STRUCT
		baseFilename : STRING[20];
		description : STRING[80];
		author : STRING[40];
		printOwner : STRING[40];
		buildInstanceID : STRING[40];
		configEditorBranch : STRING[20];
		configEditorVersion : STRING[20];
		rasterEngineBranch : STRING[20];
		rasterEngineVersion : STRING[20];
		buildLayout : UDINT;
		printNumber : UINT;
		numberOfLayers : UINT;
		layerHeight : REAL;
		encoderTickWidth : REAL;
		maxLaserCount : UINT;
		laserLineAngle : REAL;
		headCenterOffset : REAL;
		laserSpacing : REAL;
		minLaserWatts : REAL;
		maxLaserWatts : REAL;
		buildPlatformName : STRING[20];
		currentPartHeight : REAL;
		nextLayerNumber : UINT;
		currentLayerNumber : UINT;
		lastRecoatedLayerNumber : UINT;
		lastPrintedLayerNumber : UINT;
		buildInfoCheckValid : BOOL;
		newBuildInfoFileLoaded : BOOL;
		buildIteration : UINT;
		openAndCloseLayers : BOOL;
		cleanerEngagedToScoops : BOOL;
		pixelMapFileVersion : UINT;
		lastDistributedLayer : UINT;
	END_STRUCT;
END_TYPE
```

### Program Logical/DataManagement/PrintJobManagement/RM_BuildInfo (IEC) - Build Info Recipe management operations

#### Main.st
```iecst
PROGRAM _INIT

	gOpcData_ToBuildPC.Heartbeat := 0;
	gOpcData_FromBuildPC.Heartbeat := 0;

	//gOpcData_ToVisionPC.HeartbeatOut := 0;
	//gOpcData_FromVisionPC.HeartbeatIn := 0;

	gBuildInformation.base_filename := 'VF-99999-9999';
	gBuildInformation.build_iter := 0;
	gBuildInformation.description := 'n/a';
	gBuildInformation.build_layout := 99999;
	gBuildInformation.print_number := 9999;
	gBuildInformation.num_layers := 1;
	gBuildInformation.layer_height := 0.05;
	gBuildInformation.platform_id := 3;
	gBuildInformation.description := '';
	gBuildInformation.author := '';
	gBuildInformation.print_owner := '';
	gBuildInformation.platform_name := '600x600';

	gBuildInformation.build_volume_limits.min.X := 130.0;
	gBuildInformation.build_volume_limits.min.Y := 130.0;
	gBuildInformation.build_volume_limits.min.Z := 0.0;

	gBuildInformation.build_volume_limits.max.X := 728.0;
	gBuildInformation.build_volume_limits.max.Y := 728.0;
	gBuildInformation.build_volume_limits.max.Z := 400.0;

	subscribePLCOpen( gSystemRecipeApi.commands.loadBuildInfo, 'Build Info', task.commands.load, task.internal.load );

	task.internal.loaded := gSystemRecipeApi.events.buildInfoLoaded;

	registerStateBool( gPrintJobManagement.status.buildInfoInvalid, 'File Not Loaded', task.internal.notLoaded);

	task.internal.notLoaded := TRUE;

END_PROGRAM

PROGRAM _CYCLIC

	// Get the current date/time for save operations.
	fbDTGetTime.enable := TRUE;
	fbDTGetTime();
	saveTime := fbDTGetTime.DT1;

	// ---------------------------------------------------------------------------
	// BuildInfo recipe file management.
	// ---------------------------------------------------------------------------
	IF task.status.state = STATE_READY THEN

		// Prevent simultaneous load and save commands.
		//If both are true, cancel them both..
		IF (task.commands.load AND task.commands.save) THEN

			//task.internal.save.status := ERR_INHIBITED;
			//task.internal.load.status := ERR_INHIBITED;

			//vfAlarmEdgeSnippet( gPrintJobManagement.alarms.components, gPrintJobManagement.alarms.Inhibited_AL0022, 'Load and Save commanded at the same time');

		ELSIF task.commands.load THEN

			task.status.state:= STATE_LOAD;

		ELSIF task.commands.save THEN

			task.commands.save := FALSE;
			task.status.state:= STATE_SAVE;

		END_IF
	ELSE

		//TODO: Should we allow this?
		//Respond error to commands that come in while we are busy
		//Currently, this will allow commands to be saved
		//and processed when they are complete
		IF task.commands.load THEN
//			task.internal.load.status := ERR_INHIBITED;
		END_IF

		IF task.commands.load THEN
//			task.internal.save.status := ERR_INHIBITED;
		END_IF

	END_IF

	CASE task.status.state OF
		STATE_LOAD:
			fbRecipeXml_BuildInfo.Enable := TRUE;
			fbRecipeXml_BuildInfo.Load := TRUE;

			IF fbRecipeXml_BuildInfo.CommandDone THEN
				fbRecipeXml_BuildInfo.Enable := FALSE;

				task.internal.notLoaded := FALSE;
			    gSystemRecipeApi.status.buildInfoLoaded := TRUE;
				task.status.state := STATE_READY;
				task.internal.load.status := ERR_OK;
				task.commands.load := FALSE;
				//executeCommand( task.internal.loaded );

			ELSIF fbRecipeXml_BuildInfo.Error THEN

				task.internal.notLoaded := TRUE;

				fbRecipeXml_BuildInfo.ErrorReset	:= TRUE;
				fbRecipeXml_BuildInfo.Enable := FALSE;
				task.internal.load.status := PRINT_JOB_MANAGER_ERROR;
				task.status.state := STATE_READY;

				//brsitoa(fbRecipeXml_BuildInfo.StatusID, ADR(gPrintJobManagement.alarms.FileLoadError_AL0023.snippet));
				//vfAlarmEdge( gPrintJobManagement.alarms.components, gPrintJobManagement.alarms.FileLoadError_AL0023);

			END_IF

		STATE_SAVE:

			fbRecipeXml_BuildInfo.Save := TRUE;

			IF fbRecipeXml_BuildInfo.CommandDone THEN

				task.status.state := STATE_READY;
				task.internal.save.status := ERR_OK;

			ELSIF fbRecipeXml_BuildInfo.Error THEN

				fbRecipeXml_BuildInfo.ErrorReset	:= TRUE;
				task.internal.save.status := PRINT_JOB_MANAGER_ERROR;
				task.status.state := STATE_READY;

				//brsitoa( fbRecipeXml_BuildInfo.StatusID, ADR(gPrintJobManagement.alarms.FileSaveError_AL0024.snippet));
				//vfAlarmEdge( gPrintJobManagement.alarms.components, gPrintJobManagement.alarms.FileSaveError_AL0024);

			END_IF

	END_CASE

	fbRecipeXml_BuildInfo.MpLink := ADR(gBuildInfoRecipe);
	fbRecipeXml_BuildInfo.DeviceName := ADR('CurrentBuild');
	fbRecipeXml_BuildInfo.Category := ADR('BuildInfo');
	fbRecipeXml_BuildInfo.FileName := ADR('BuildInfo.xml');
	//fbRecipeXml_BuildInfo.Header := ADR(header_BuildInfo);  // BuildInfo.xml file has no header
	fbRecipeXml_BuildInfo.LoadType := mpRECIPE_XML_LOAD_ALL;
	fbRecipeXml_BuildInfo();
	fbRecipeXml_BuildInfo.Save := FALSE;
	fbRecipeXml_BuildInfo.Load := FALSE;
	fbRecipeXml_BuildInfo.ErrorReset := FALSE;

	fbRecipeRegPar_BuildInfo.MpLink := ADR(gBuildInfoRecipe);
	fbRecipeRegPar_BuildInfo.Enable := TRUE;
	fbRecipeRegPar_BuildInfo.PVName := ADR('gBuildInformation');
	fbRecipeRegPar_BuildInfo.Category := ADR('BuildInfo');
	fbRecipeRegPar_BuildInfo();
	fbRecipeRegPar_BuildInfo.ErrorReset := FALSE;

	//If we are not ready, and the build info IS ready, go to ready
	IF task.status.state =  STATE_NOT_READY AND fbRecipeRegPar_BuildInfo.StatusID = ERR_OK THEN

		task.status.state:= STATE_READY;

	END_IF

	// Update the command status; if an error occurs, update select the first applicable status ID.
	task.status.busy := fbRecipeXml_BuildInfo.CommandBusy;
	task.status.done := fbRecipeXml_BuildInfo.CommandDone;
	task.status.error := fbRecipeRegPar_BuildInfo.Error OR fbRecipeXml_BuildInfo.Error;
	IF (fbRecipeRegPar_BuildInfo.Error) THEN
		task.status.errorId := fbRecipeRegPar_BuildInfo.StatusID;
	ELSIF (fbRecipeXml_BuildInfo.Error) THEN
		task.status.errorId := fbRecipeXml_BuildInfo.StatusID;
	ELSE
		task.status.errorId := ERR_OK;
	END_IF

END_PROGRAM

PROGRAM _EXIT

	// Prevent error mpRECIPE_ERR_MPLINK_IN_USE by releasing the link to the configuration objects.
	fbRecipeRegPar_BuildInfo.Enable := FALSE;
	fbRecipeRegPar_BuildInfo();
	fbRecipeXml_BuildInfo.Enable := FALSE;
	fbRecipeXml_BuildInfo();

END_PROGRAM
```

### Program Logical/DataManagement/PrintJobManagement/RM_PrintProcessConfig (IEC)

#### Types.typ
```iecst
TYPE
	PrintProcessConfigTask_typ : 	STRUCT
		commands : PrintConfigCommands_typ;
		parameters : PrintConfigParameters_typ;
		status : PrintConfigStatus_typ;
		internal : PrintConfigInternal_typ;
	END_STRUCT;
	PrintConfigCommands_typ : 	STRUCT
		load : BOOL;
		save : BOOL;
	END_STRUCT;
	PrintConfigParameters_typ : 	STRUCT
		_ : STRING[260];
	END_STRUCT;
	PrintConfigStatus_typ : 	STRUCT
		state : STATE;
		busy : BOOL;
		done : BOOL;
		error : BOOL;
		errorId : DINT;
		loadPCIComplete : BOOL;
		pciLoadStatus : STRING[12];
	END_STRUCT;
	PrintConfigInternal_typ : 	STRUCT
		save : AtnPlcOpenStatus;
		load : AtnPlcOpenStatus;
		enableManualOverwrite : BOOL;
		_previousPciLoaded : BOOL;
		atnCommand : AtnPLCOpen;
		hmiSelectedPciParameterData : HMISelectedPciParData_typ;
		_previousOverwriteStatus : BOOL;
	END_STRUCT;
	HMIInputs_typ : 	STRUCT
		ContinuousModeEnable : BOOL;
		ContinuousModeDisable : BOOL;
		GasFlowLpm : REAL;
		RecSpreadVelocity : REAL;
		RecSpreadAccel : REAL;
		RecSpreadDecel : REAL;
		RecApproachVelocity : REAL;
		RecApproachAccel : REAL;
		RecApproachDecel : REAL;
		ElectrodeEnable : BOOL;
		ElectrodeDisable : BOOL;
		ElectrodeGainPerc : REAL;
		MhInitialDispenseRot : REAL;
		MhContinuousDispenseRot : REAL;
		AiMaxRecoatLimit : REAL;
		ApplyRecSpreadVel : BOOL;
		ApplyRecApproachVel : BOOL;
		ApplyGasFlow : BOOL;
		ApplyElectrodeGain : BOOL;
		ApplyInitialDispenseRot : BOOL;
		ApplyContDispenseRot : BOOL;
		ApplyAiMaxRecoatLimit : BOOL;
		DropdownSelection : USINT;
	END_STRUCT;
	HMISelectedPciParData_typ : 	STRUCT
		MachineName : STRING[5];
		Description : STRING[255];
		FileFormatVersion : INT;
		DateTimeGenerated : STRING[30];
		ParamterSetpoints : ParamterSetpoints_typ;
	END_STRUCT;
	STATE :
		(
		STATE_NOT_READY,
		STATE_READY,
		STATE_DONE,
		STATE_ERROR,
		STATE_LOAD,
		STATE_SAVE
		);
END_TYPE
```

#### Variables.var
```iecst
VAR
	fbRecipeXml_PrintProcessConfig : MpRecipeXml := (0);
	fbRecipeRegPar_PrintConfig : MpRecipeRegPar := (0);
	task : PrintProcessConfigTask_typ;
	HMIInputs : HMIInputs_typ;
	ii : USINT; (*Loop Var*)
	jj : USINT; (*Loop Var*)
	gPrintProcessConfigRecipe : {REDUND_UNREPLICABLE} MpComIdentType; (*#1"C:\ControlPLC_Gen3_Rev0\Gen3\ControlPLC_Gen3_Rev0\Physical\ControlPLC_Gen3\5PC900_TS17_02\mappServices\Recipies.mprecipexml" #2"1" #3"1"*)
END_VAR
```

#### Cyclic.st
```iecst
PROGRAM _CYCLIC

	// ---------------------------------------------------------------------------
	// PrintProcessConfig recipe file management.
	// ---------------------------------------------------------------------------

	IF task.status.state = STATE_READY THEN

		IF  task.commands.load THEN

			task.status.state:= STATE_LOAD;

		END_IF

	ELSE

		//TODO: Should we allow this?
		//Respond error to commands that come in while we are busy
		//Currently, this will allow commands to be saved
		//and processed when they are complete
		IF task.commands.load THEN
			//			task.internal.load.status := ERR_INHIBITED;
		END_IF

		IF task.commands.load THEN
			//			task.internal.save.status := ERR_INHIBITED;
		END_IF

	END_IF

	CASE task.status.state OF

		STATE_LOAD:

			fbRecipeXml_PrintProcessConfig.Load := TRUE;

			IF fbRecipeXml_PrintProcessConfig.CommandDone THEN

				gPrintJobManagement.status.loadPCIFileComplete := TRUE;

				task.internal.load.status := ERR_OK;

				task.status.state := STATE_READY;

			ELSIF fbRecipeXml_PrintProcessConfig.Error THEN

				fbRecipeXml_PrintProcessConfig.ErrorReset	:= TRUE;
				task.internal.load.status := PRINT_JOB_MANAGER_ERROR;

				task.status.state := STATE_READY;

				//brsitoa(fbRecipeXml_PrintProcessConfig.StatusID, ADR(gPrintJobManagement.alarms.FileLoadError_AL0023.snippet));
				//vfAlarmEdge( gPrintJobManagement.alarms.components, gPrintJobManagement.alarms.FileLoadError_AL0023);

			END_IF

		STATE_SAVE:

			fbRecipeXml_PrintProcessConfig.Save := TRUE;

			IF fbRecipeXml_PrintProcessConfig.CommandDone THEN

				task.status.state := STATE_READY;
				task.internal.save.status := ERR_OK;

			ELSIF fbRecipeXml_PrintProcessConfig.Error THEN

				fbRecipeXml_PrintProcessConfig.ErrorReset	:= TRUE;
				task.internal.save.status := PRINT_JOB_MANAGER_ERROR;
				task.status.state := STATE_READY;

				//brsitoa( fbRecipeXml_PrintProcessConfig.StatusID, ADR(gPrintJobManagement.alarms.FileSaveError_AL0024.snippet));
				//vfAlarmEdge( gPrintJobManagement.alarms.components, gPrintJobManagement.alarms.FileSaveError_AL0024);

			END_IF

	END_CASE

	task.commands.load := FALSE;
	task.commands.save := FALSE;

	//RECIPE FOR LOADING AND SAVING THE MEASUREMENT LOCATIONS
	fbRecipeXml_PrintProcessConfig.MpLink := ADR(gPrintProcessConfigRecipe);
	fbRecipeXml_PrintProcessConfig.Enable := TRUE;
	fbRecipeXml_PrintProcessConfig.DeviceName := ADR('CurrentBuild');
	fbRecipeXml_PrintProcessConfig.Category := ADR('CurrentBuild');
	fbRecipeXml_PrintProcessConfig.FileName := ADR('PrintProcessConfig.xml');
	//fbRecipeXml_PrintProcessConfig.Header := ADR(header_CustomScan);  // CustomScan.xml file has no header
	fbRecipeXml_PrintProcessConfig.LoadType := mpRECIPE_XML_LOAD_ALL;
	fbRecipeXml_PrintProcessConfig();
	fbRecipeXml_PrintProcessConfig.Save := FALSE;
	fbRecipeXml_PrintProcessConfig.Load := FALSE;
	fbRecipeXml_PrintProcessConfig.ErrorReset := FALSE;

	fbRecipeRegPar_PrintConfig.MpLink := ADR(gPrintProcessConfigRecipe);
	fbRecipeRegPar_PrintConfig.Enable := TRUE;
	fbRecipeRegPar_PrintConfig.PVName := ADR('gPrintProcessConfig');
	fbRecipeRegPar_PrintConfig.Category := ADR('CurrentBuild');
	fbRecipeRegPar_PrintConfig();
	fbRecipeRegPar_PrintConfig.ErrorReset := FALSE;

	//If we are not ready, and the build info IS ready, go to ready
	IF task.status.state =  STATE_NOT_READY AND fbRecipeRegPar_PrintConfig.StatusID = ERR_OK THEN

		task.status.state:= STATE_READY;

	END_IF

	// Update the command status; if an error occurs, update select the first applicable status ID.
	task.status.busy := fbRecipeXml_PrintProcessConfig.CommandBusy;
	task.status.done := fbRecipeXml_PrintProcessConfig.CommandDone;
	task.status.error := fbRecipeRegPar_PrintConfig.Error OR fbRecipeXml_PrintProcessConfig.Error;
	IF (fbRecipeRegPar_PrintConfig.Error) THEN
		task.status.errorId := fbRecipeRegPar_PrintConfig.StatusID;
	ELSIF (fbRecipeXml_PrintProcessConfig.Error) THEN
		task.status.errorId := fbRecipeXml_PrintProcessConfig.StatusID;
	ELSE
		task.status.errorId := ERR_OK;

	END_IF

	DeriveProcessData;

END_PROGRAM
```

#### DeriveProcessData.st
```iecst
ACTION DeriveProcessData:

	// ATN command handle
	task.internal.atnCommand();
	IF task.internal.atnCommand.Done OR task.internal.atnCommand.Error OR task.internal.atnCommand.Aborted THEN
		task.internal.atnCommand.Execute := FALSE;
	END_IF

	// ==================================================================================================================================================

	IF gPrintProcessConfigLoaded THEN
		task.status.pciLoadStatus := 'LOADED';
	ELSE
		task.status.pciLoadStatus := 'NOT LOADED';
	END_IF

END_ACTION
```

#### Exit.st
```iecst
PROGRAM _EXIT

	// Prevent error mpRECIPE_ERR_MPLINK_IN_USE by releasing the link to the configuration objects.
	fbRecipeXml_PrintProcessConfig.Enable := FALSE;
	fbRecipeXml_PrintProcessConfig();

END_PROGRAM
```

### Program Logical/DataManagement/PrintJobManagement/PrintJobManagement (IEC) - Print job management operations
